(* Logix 5000 project; controller QW361 vendor 1 type 14 code 107 rev 32.11; software revision 32.00; part 8 of 20 *)

        [856].log_data[0].maxminute := 50, [856].log_data[0].valid := 1, [856].log_data[1].valid := 1, [856].log_data[2].valid := 1, [856].log_data[3].valid := 1, [856].log_data[4].valid := 1, [856].time.Year := 2022, [856].time.Month := 4, [856].time.Day := 26, [856].time.Hour := 20, [856].time.Minute := 54, [856].time.Second := 59, [856].time.DST_ON := 1, [857].log_data[0].min := 1.0, [857].log_data[0].max := 1.0, [857].log_data[0].total := 299.999, [857].log_data[0].time := 299.999, [857].log_data[0].minminute := 55, [857].log_data[0].maxminute := 55, [857].log_data[0].valid := 1, [857].log_data[1].valid := 1, [857].log_data[2].valid := 1, [857].log_data[3].valid := 1, [857].log_data[4].valid := 1, [857].time.Year := 2022, [857].time.Month := 4, [857].time.Day := 26, [857].time.Hour := 20, [857].time.Minute := 59, [857].time.Second := 59, [857].time.DST_ON := 1, [858].log_data[0].min := 1.0, [858].log_data[0].max := 1.0, [858].log_data[0].total := 300.0, [858].log_data[0].time := 300.0, [858].log_data[0].valid := 1, [858].log_data[1].valid := 1, [858].log_data[2].valid := 1, [858].log_data[3].valid := 1, [858].log_data[4].valid := 1, [858].time.Year := 2022, [858].time.Month := 4, [858].time.Day := 26, [858].time.Hour := 21, [858].time.Minute := 4, [858].time.Second := 59, [858].time.DST_ON := 1, [859].log_data[0].min := 1.0, [859].log_data[0].max := 1.0, [859].log_data[0].total := 300.0, [859].log_data[0].time := 300.0, [859].log_data[0].minminute := 5, [859].log_data[0].maxminute := 5, [859].log_data[0].valid := 1, [859].log_data[1].valid := 1, [859].log_data[2].valid := 1, [859].log_data[3].valid := 1, [859].log_data[4].valid := 1, [859].time.Year := 2022, [859].time.Month := 4,
        [859].time.Day := 26, [859].time.Hour := 21, [859].time.Minute := 9, [859].time.Second := 59, [859].time.DST_ON := 1, [860].log_data[0].min := 1.0, [860].log_data[0].max := 1.0, [860].log_data[0].total := 300.0, [860].log_data[0].time := 300.0, [860].log_data[0].minminute := 10, [860].log_data[0].maxminute := 10, [860].log_data[0].valid := 1, [860].log_data[1].valid := 1, [860].log_data[2].valid := 1, [860].log_data[3].valid := 1, [860].log_data[4].valid := 1, [860].time.Year := 2022, [860].time.Month := 4, [860].time.Day := 26, [860].time.Hour := 21, [860].time.Minute := 14, [860].time.Second := 59, [860].time.DST_ON := 1, [861].log_data[0].min := 1.0, [861].log_data[0].max := 1.0, [861].log_data[0].total := 300.0, [861].log_data[0].time := 300.0, [861].log_data[0].minminute := 15, [861].log_data[0].maxminute := 15, [861].log_data[0].valid := 1, [861].log_data[1].valid := 1, [861].log_data[2].valid := 1, [861].log_data[3].valid := 1, [861].log_data[4].valid := 1, [861].time.Year := 2022, [861].time.Month := 4, [861].time.Day := 26, [861].time.Hour := 21, [861].time.Minute := 19, [861].time.Second := 59, [861].time.DST_ON := 1, [862].log_data[0].min := 1.0, [862].log_data[0].max := 1.0, [862].log_data[0].total := 300.0, [862].log_data[0].time := 300.0, [862].log_data[0].minminute := 20, [862].log_data[0].maxminute := 20, [862].log_data[0].valid := 1, [862].log_data[1].valid := 1, [862].log_data[2].valid := 1, [862].log_data[3].valid := 1, [862].log_data[4].valid := 1, [862].time.Year := 2022, [862].time.Month := 4, [862].time.Day := 26, [862].time.Hour := 21, [862].time.Minute := 24, [862].time.Second := 59, [862].time.DST_ON := 1, [863].log_data[0].min := 1.0,
        [863].log_data[0].max := 1.0, [863].log_data[0].total := 300.0, [863].log_data[0].time := 300.0, [863].log_data[0].minminute := 25, [863].log_data[0].maxminute := 25, [863].log_data[0].valid := 1, [863].log_data[1].valid := 1, [863].log_data[2].valid := 1, [863].log_data[3].valid := 1, [863].log_data[4].valid := 1, [863].time.Year := 2022, [863].time.Month := 4, [863].time.Day := 26, [863].time.Hour := 21, [863].time.Minute := 29, [863].time.Second := 59, [863].time.DST_ON := 1, [864].log_data[0].min := 1.0, [864].log_data[0].max := 1.0, [864].log_data[0].total := 300.0, [864].log_data[0].time := 300.0, [864].log_data[0].minminute := 30, [864].log_data[0].maxminute := 30, [864].log_data[0].valid := 1, [864].log_data[1].valid := 1, [864].log_data[2].valid := 1, [864].log_data[3].valid := 1, [864].log_data[4].valid := 1, [864].time.Year := 2022, [864].time.Month := 4, [864].time.Day := 26, [864].time.Hour := 21, [864].time.Minute := 34, [864].time.Second := 59, [864].time.DST_ON := 1, [865].log_data[0].min := 1.0, [865].log_data[0].max := 1.0, [865].log_data[0].total := 300.0, [865].log_data[0].time := 300.0, [865].log_data[0].minminute := 35, [865].log_data[0].maxminute := 35, [865].log_data[0].valid := 1, [865].log_data[1].valid := 1, [865].log_data[2].valid := 1, [865].log_data[3].valid := 1, [865].log_data[4].valid := 1, [865].time.Year := 2022, [865].time.Month := 4, [865].time.Day := 26, [865].time.Hour := 21, [865].time.Minute := 39, [865].time.Second := 59, [865].time.DST_ON := 1, [866].log_data[0].min := 1.0, [866].log_data[0].max := 1.0, [866].log_data[0].total := 300.0, [866].log_data[0].time := 300.0, [866].log_data[0].minminute := 40, [866].log_data[0].maxminute := 40, [866].log_data[0].valid := 1,
        [866].log_data[1].valid := 1, [866].log_data[2].valid := 1, [866].log_data[3].valid := 1, [866].log_data[4].valid := 1, [866].time.Year := 2022, [866].time.Month := 4, [866].time.Day := 26, [866].time.Hour := 21, [866].time.Minute := 44, [866].time.Second := 59, [866].time.DST_ON := 1, [867].log_data[0].min := 1.0, [867].log_data[0].max := 1.0, [867].log_data[0].total := 300.0, [867].log_data[0].time := 300.0, [867].log_data[0].minminute := 45, [867].log_data[0].maxminute := 45, [867].log_data[0].valid := 1, [867].log_data[1].valid := 1, [867].log_data[2].valid := 1, [867].log_data[3].valid := 1, [867].log_data[4].valid := 1, [867].time.Year := 2022, [867].time.Month := 4, [867].time.Day := 26, [867].time.Hour := 21, [867].time.Minute := 49, [867].time.Second := 59, [867].time.DST_ON := 1, [868].log_data[0].min := 1.0, [868].log_data[0].max := 1.0, [868].log_data[0].total := 300.0, [868].log_data[0].time := 300.0, [868].log_data[0].minminute := 50, [868].log_data[0].maxminute := 50, [868].log_data[0].valid := 1, [868].log_data[1].valid := 1, [868].log_data[2].valid := 1, [868].log_data[3].valid := 1, [868].log_data[4].valid := 1, [868].time.Year := 2022, [868].time.Month := 4, [868].time.Day := 26, [868].time.Hour := 21, [868].time.Minute := 54, [868].time.Second := 59, [868].time.DST_ON := 1, [869].log_data[0].min := 1.0, [869].log_data[0].max := 1.0, [869].log_data[0].total := 300.0, [869].log_data[0].time := 300.0, [869].log_data[0].minminute := 55, [869].log_data[0].maxminute := 55, [869].log_data[0].valid := 1, [869].log_data[1].valid := 1, [869].log_data[2].valid := 1, [869].log_data[3].valid := 1, [869].log_data[4].valid := 1, [869].time.Year := 2022, [869].time.Month := 4,
        [869].time.Day := 26, [869].time.Hour := 21, [869].time.Minute := 59, [869].time.Second := 59, [869].time.DST_ON := 1, [870].log_data[0].min := 1.0, [870].log_data[0].max := 1.0, [870].log_data[0].total := 300.0, [870].log_data[0].time := 300.0, [870].log_data[0].valid := 1, [870].log_data[1].valid := 1, [870].log_data[2].valid := 1, [870].log_data[3].valid := 1, [870].log_data[4].valid := 1, [870].time.Year := 2022, [870].time.Month := 4, [870].time.Day := 26, [870].time.Hour := 22, [870].time.Minute := 4, [870].time.Second := 59, [870].time.DST_ON := 1, [871].log_data[0].min := 1.0, [871].log_data[0].max := 1.0, [871].log_data[0].total := 300.0, [871].log_data[0].time := 300.0, [871].log_data[0].minminute := 5, [871].log_data[0].maxminute := 5, [871].log_data[0].valid := 1, [871].log_data[1].valid := 1, [871].log_data[2].valid := 1, [871].log_data[3].valid := 1, [871].log_data[4].valid := 1, [871].time.Year := 2022, [871].time.Month := 4, [871].time.Day := 26, [871].time.Hour := 22, [871].time.Minute := 9, [871].time.Second := 59, [871].time.DST_ON := 1, [872].log_data[0].min := 1.0, [872].log_data[0].max := 1.0, [872].log_data[0].total := 300.0, [872].log_data[0].time := 300.0, [872].log_data[0].minminute := 10, [872].log_data[0].maxminute := 10, [872].log_data[0].valid := 1, [872].log_data[1].valid := 1, [872].log_data[2].valid := 1, [872].log_data[3].valid := 1, [872].log_data[4].valid := 1, [872].time.Year := 2022, [872].time.Month := 4, [872].time.Day := 26, [872].time.Hour := 22, [872].time.Minute := 14, [872].time.Second := 59, [872].time.DST_ON := 1, [873].log_data[0].min := 1.0, [873].log_data[0].max := 1.0, [873].log_data[0].total := 300.0,
        [873].log_data[0].time := 300.0, [873].log_data[0].minminute := 15, [873].log_data[0].maxminute := 15, [873].log_data[0].valid := 1, [873].log_data[1].valid := 1, [873].log_data[2].valid := 1, [873].log_data[3].valid := 1, [873].log_data[4].valid := 1, [873].time.Year := 2022, [873].time.Month := 4, [873].time.Day := 26, [873].time.Hour := 22, [873].time.Minute := 19, [873].time.Second := 59, [873].time.DST_ON := 1, [874].log_data[0].min := 1.0, [874].log_data[0].max := 1.0, [874].log_data[0].total := 300.0, [874].log_data[0].time := 300.0, [874].log_data[0].minminute := 20, [874].log_data[0].maxminute := 20, [874].log_data[0].valid := 1, [874].log_data[1].valid := 1, [874].log_data[2].valid := 1, [874].log_data[3].valid := 1, [874].log_data[4].valid := 1, [874].time.Year := 2022, [874].time.Month := 4, [874].time.Day := 26, [874].time.Hour := 22, [874].time.Minute := 24, [874].time.Second := 59, [874].time.DST_ON := 1, [875].log_data[0].min := 1.0, [875].log_data[0].max := 1.0, [875].log_data[0].total := 300.0, [875].log_data[0].time := 300.0, [875].log_data[0].minminute := 25, [875].log_data[0].maxminute := 25, [875].log_data[0].valid := 1, [875].log_data[1].valid := 1, [875].log_data[2].valid := 1, [875].log_data[3].valid := 1, [875].log_data[4].valid := 1, [875].time.Year := 2022, [875].time.Month := 4, [875].time.Day := 26, [875].time.Hour := 22, [875].time.Minute := 29, [875].time.Second := 59, [875].time.DST_ON := 1, [876].log_data[0].min := 1.0, [876].log_data[0].max := 1.0, [876].log_data[0].total := 300.0, [876].log_data[0].time := 300.0, [876].log_data[0].minminute := 30, [876].log_data[0].maxminute := 30, [876].log_data[0].valid := 1, [876].log_data[1].valid := 1, [876].log_data[2].valid := 1,
        [876].log_data[3].valid := 1, [876].log_data[4].valid := 1, [876].time.Year := 2022, [876].time.Month := 4, [876].time.Day := 26, [876].time.Hour := 22, [876].time.Minute := 34, [876].time.Second := 59, [876].time.DST_ON := 1, [877].log_data[0].min := 1.0, [877].log_data[0].max := 1.0, [877].log_data[0].total := 300.0, [877].log_data[0].time := 300.0, [877].log_data[0].minminute := 35, [877].log_data[0].maxminute := 35, [877].log_data[0].valid := 1, [877].log_data[1].valid := 1, [877].log_data[2].valid := 1, [877].log_data[3].valid := 1, [877].log_data[4].valid := 1, [877].time.Year := 2022, [877].time.Month := 4, [877].time.Day := 26, [877].time.Hour := 22, [877].time.Minute := 39, [877].time.Second := 59, [877].time.DST_ON := 1, [878].log_data[0].min := 1.0, [878].log_data[0].max := 1.0, [878].log_data[0].total := 300.0, [878].log_data[0].time := 300.0, [878].log_data[0].minminute := 40, [878].log_data[0].maxminute := 40, [878].log_data[0].valid := 1, [878].log_data[1].valid := 1, [878].log_data[2].valid := 1, [878].log_data[3].valid := 1, [878].log_data[4].valid := 1, [878].time.Year := 2022, [878].time.Month := 4, [878].time.Day := 26, [878].time.Hour := 22, [878].time.Minute := 44, [878].time.Second := 59, [878].time.DST_ON := 1, [879].log_data[0].min := 1.0, [879].log_data[0].max := 1.0, [879].log_data[0].total := 300.0, [879].log_data[0].time := 300.0, [879].log_data[0].minminute := 45, [879].log_data[0].maxminute := 45, [879].log_data[0].valid := 1, [879].log_data[1].valid := 1, [879].log_data[2].valid := 1, [879].log_data[3].valid := 1, [879].log_data[4].valid := 1, [879].time.Year := 2022, [879].time.Month := 4, [879].time.Day := 26, [879].time.Hour := 22,
        [879].time.Minute := 49, [879].time.Second := 59, [879].time.DST_ON := 1, [880].log_data[0].min := 1.0, [880].log_data[0].max := 1.0, [880].log_data[0].total := 300.0, [880].log_data[0].time := 300.0, [880].log_data[0].minminute := 50, [880].log_data[0].maxminute := 50, [880].log_data[0].valid := 1, [880].log_data[1].valid := 1, [880].log_data[2].valid := 1, [880].log_data[3].valid := 1, [880].log_data[4].valid := 1, [880].time.Year := 2022, [880].time.Month := 4, [880].time.Day := 26, [880].time.Hour := 22, [880].time.Minute := 54, [880].time.Second := 59, [880].time.DST_ON := 1, [881].log_data[0].min := 1.0, [881].log_data[0].max := 1.0, [881].log_data[0].total := 300.0, [881].log_data[0].time := 300.0, [881].log_data[0].minminute := 55, [881].log_data[0].maxminute := 55, [881].log_data[0].valid := 1, [881].log_data[1].valid := 1, [881].log_data[2].valid := 1, [881].log_data[3].valid := 1, [881].log_data[4].valid := 1, [881].time.Year := 2022, [881].time.Month := 4, [881].time.Day := 26, [881].time.Hour := 22, [881].time.Minute := 59, [881].time.Second := 59, [881].time.DST_ON := 1, [882].log_data[0].min := 1.0, [882].log_data[0].max := 1.0, [882].log_data[0].total := 300.0, [882].log_data[0].time := 300.0, [882].log_data[0].valid := 1, [882].log_data[1].valid := 1, [882].log_data[2].valid := 1, [882].log_data[3].valid := 1, [882].log_data[4].valid := 1, [882].time.Year := 2022, [882].time.Month := 4, [882].time.Day := 26, [882].time.Hour := 23, [882].time.Minute := 4, [882].time.Second := 59, [882].time.DST_ON := 1, [883].log_data[0].min := 1.0, [883].log_data[0].max := 1.0, [883].log_data[0].total := 300.0, [883].log_data[0].time := 300.0, [883].log_data[0].minminute := 5,
        [883].log_data[0].maxminute := 5, [883].log_data[0].valid := 1, [883].log_data[1].valid := 1, [883].log_data[2].valid := 1, [883].log_data[3].valid := 1, [883].log_data[4].valid := 1, [883].time.Year := 2022, [883].time.Month := 4, [883].time.Day := 26, [883].time.Hour := 23, [883].time.Minute := 9, [883].time.Second := 59, [883].time.DST_ON := 1, [884].log_data[0].min := 1.0, [884].log_data[0].max := 1.0, [884].log_data[0].total := 300.0, [884].log_data[0].time := 300.0, [884].log_data[0].minminute := 10, [884].log_data[0].maxminute := 10, [884].log_data[0].valid := 1, [884].log_data[1].valid := 1, [884].log_data[2].valid := 1, [884].log_data[3].valid := 1, [884].log_data[4].valid := 1, [884].time.Year := 2022, [884].time.Month := 4, [884].time.Day := 26, [884].time.Hour := 23, [884].time.Minute := 14, [884].time.Second := 59, [884].time.DST_ON := 1, [885].log_data[0].min := 1.0, [885].log_data[0].max := 1.0, [885].log_data[0].total := 300.0, [885].log_data[0].time := 300.0, [885].log_data[0].minminute := 15, [885].log_data[0].maxminute := 15, [885].log_data[0].valid := 1, [885].log_data[1].valid := 1, [885].log_data[2].valid := 1, [885].log_data[3].valid := 1, [885].log_data[4].valid := 1, [885].time.Year := 2022, [885].time.Month := 4, [885].time.Day := 26, [885].time.Hour := 23, [885].time.Minute := 19, [885].time.Second := 59, [885].time.DST_ON := 1, [886].log_data[0].min := 1.0, [886].log_data[0].max := 1.0, [886].log_data[0].total := 300.0, [886].log_data[0].time := 300.0, [886].log_data[0].minminute := 20, [886].log_data[0].maxminute := 20, [886].log_data[0].valid := 1, [886].log_data[1].valid := 1, [886].log_data[2].valid := 1, [886].log_data[3].valid := 1, [886].log_data[4].valid := 1,
        [886].time.Year := 2022, [886].time.Month := 4, [886].time.Day := 26, [886].time.Hour := 23, [886].time.Minute := 24, [886].time.Second := 59, [886].time.DST_ON := 1, [887].log_data[0].min := 1.0, [887].log_data[0].max := 1.0, [887].log_data[0].total := 300.0, [887].log_data[0].time := 300.0, [887].log_data[0].minminute := 25, [887].log_data[0].maxminute := 25, [887].log_data[0].valid := 1, [887].log_data[1].valid := 1, [887].log_data[2].valid := 1, [887].log_data[3].valid := 1, [887].log_data[4].valid := 1, [887].time.Year := 2022, [887].time.Month := 4, [887].time.Day := 26, [887].time.Hour := 23, [887].time.Minute := 29, [887].time.Second := 59, [887].time.DST_ON := 1, [888].log_data[0].min := 1.0, [888].log_data[0].max := 1.0, [888].log_data[0].total := 300.0, [888].log_data[0].time := 300.0, [888].log_data[0].minminute := 30, [888].log_data[0].maxminute := 30, [888].log_data[0].valid := 1, [888].log_data[1].valid := 1, [888].log_data[2].valid := 1, [888].log_data[3].valid := 1, [888].log_data[4].valid := 1, [888].time.Year := 2022, [888].time.Month := 4, [888].time.Day := 26, [888].time.Hour := 23, [888].time.Minute := 34, [888].time.Second := 59, [888].time.DST_ON := 1, [889].log_data[0].min := 1.0, [889].log_data[0].max := 1.0, [889].log_data[0].total := 300.0, [889].log_data[0].time := 300.0, [889].log_data[0].minminute := 35, [889].log_data[0].maxminute := 35, [889].log_data[0].valid := 1, [889].log_data[1].valid := 1, [889].log_data[2].valid := 1, [889].log_data[3].valid := 1, [889].log_data[4].valid := 1, [889].time.Year := 2022, [889].time.Month := 4, [889].time.Day := 26, [889].time.Hour := 23, [889].time.Minute := 39, [889].time.Second := 59,
        [889].time.DST_ON := 1, [890].log_data[0].min := 1.0, [890].log_data[0].max := 1.0, [890].log_data[0].total := 300.0, [890].log_data[0].time := 300.0, [890].log_data[0].minminute := 40, [890].log_data[0].maxminute := 40, [890].log_data[0].valid := 1, [890].log_data[1].valid := 1, [890].log_data[2].valid := 1, [890].log_data[3].valid := 1, [890].log_data[4].valid := 1, [890].time.Year := 2022, [890].time.Month := 4, [890].time.Day := 26, [890].time.Hour := 23, [890].time.Minute := 44, [890].time.Second := 59, [890].time.DST_ON := 1, [891].log_data[0].min := 1.0, [891].log_data[0].max := 1.0, [891].log_data[0].total := 300.0, [891].log_data[0].time := 300.0, [891].log_data[0].minminute := 45, [891].log_data[0].maxminute := 45, [891].log_data[0].valid := 1, [891].log_data[1].valid := 1, [891].log_data[2].valid := 1, [891].log_data[3].valid := 1, [891].log_data[4].valid := 1, [891].time.Year := 2022, [891].time.Month := 4, [891].time.Day := 26, [891].time.Hour := 23, [891].time.Minute := 49, [891].time.Second := 59, [891].time.DST_ON := 1, [892].log_data[0].min := 1.0, [892].log_data[0].max := 1.0, [892].log_data[0].total := 300.0, [892].log_data[0].time := 300.0, [892].log_data[0].minminute := 50, [892].log_data[0].maxminute := 50, [892].log_data[0].valid := 1, [892].log_data[1].valid := 1, [892].log_data[2].valid := 1, [892].log_data[3].valid := 1, [892].log_data[4].valid := 1, [892].time.Year := 2022, [892].time.Month := 4, [892].time.Day := 26, [892].time.Hour := 23, [892].time.Minute := 54, [892].time.Second := 59, [892].time.DST_ON := 1, [893].log_data[0].min := 1.0, [893].log_data[0].max := 1.0, [893].log_data[0].total := 299.999, [893].log_data[0].time := 299.999, [893].log_data[0].minminute := 55,
        [893].log_data[0].maxminute := 55, [893].log_data[0].valid := 1, [893].log_data[1].valid := 1, [893].log_data[2].valid := 1, [893].log_data[3].valid := 1, [893].log_data[4].valid := 1, [893].time.Year := 2022, [893].time.Month := 4, [893].time.Day := 26, [893].time.Hour := 23, [893].time.Minute := 59, [893].time.Second := 59, [893].time.DST_ON := 1, [894].log_data[0].min := 1.0, [894].log_data[0].max := 1.0, [894].log_data[0].total := 300.0, [894].log_data[0].time := 300.0, [894].log_data[0].valid := 1, [894].log_data[1].valid := 1, [894].log_data[2].valid := 1, [894].log_data[3].valid := 1, [894].log_data[4].valid := 1, [894].time.Year := 2022, [894].time.Month := 4, [894].time.Day := 27, [894].time.Minute := 4, [894].time.Second := 59, [894].time.DST_ON := 1, [895].log_data[0].min := 1.0, [895].log_data[0].max := 1.0, [895].log_data[0].total := 300.0, [895].log_data[0].time := 300.0, [895].log_data[0].minminute := 5, [895].log_data[0].maxminute := 5, [895].log_data[0].valid := 1, [895].log_data[1].valid := 1, [895].log_data[2].valid := 1, [895].log_data[3].valid := 1, [895].log_data[4].valid := 1, [895].time.Year := 2022, [895].time.Month := 4, [895].time.Day := 27, [895].time.Minute := 9, [895].time.Second := 59, [895].time.DST_ON := 1, [896].log_data[0].min := 1.0, [896].log_data[0].max := 1.0, [896].log_data[0].total := 300.0, [896].log_data[0].time := 300.0, [896].log_data[0].minminute := 10, [896].log_data[0].maxminute := 10, [896].log_data[0].valid := 1, [896].log_data[1].valid := 1, [896].log_data[2].valid := 1, [896].log_data[3].valid := 1, [896].log_data[4].valid := 1, [896].time.Year := 2022, [896].time.Month := 4, [896].time.Day := 27, [896].time.Minute := 14,
        [896].time.Second := 59, [896].time.DST_ON := 1, [897].log_data[0].min := 1.0, [897].log_data[0].max := 1.0, [897].log_data[0].total := 300.0, [897].log_data[0].time := 300.0, [897].log_data[0].minminute := 15, [897].log_data[0].maxminute := 15, [897].log_data[0].valid := 1, [897].log_data[1].valid := 1, [897].log_data[2].valid := 1, [897].log_data[3].valid := 1, [897].log_data[4].valid := 1, [897].time.Year := 2022, [897].time.Month := 4, [897].time.Day := 27, [897].time.Minute := 19, [897].time.Second := 59, [897].time.DST_ON := 1, [898].log_data[0].min := 1.0, [898].log_data[0].max := 1.0, [898].log_data[0].total := 300.0, [898].log_data[0].time := 300.0, [898].log_data[0].minminute := 20, [898].log_data[0].maxminute := 20, [898].log_data[0].valid := 1, [898].log_data[1].valid := 1, [898].log_data[2].valid := 1, [898].log_data[3].valid := 1, [898].log_data[4].valid := 1, [898].time.Year := 2022, [898].time.Month := 4, [898].time.Day := 27, [898].time.Minute := 24, [898].time.Second := 59, [898].time.DST_ON := 1, [899].log_data[0].min := 1.0, [899].log_data[0].max := 1.0, [899].log_data[0].total := 300.0, [899].log_data[0].time := 300.0, [899].log_data[0].minminute := 25, [899].log_data[0].maxminute := 25, [899].log_data[0].valid := 1, [899].log_data[1].valid := 1, [899].log_data[2].valid := 1, [899].log_data[3].valid := 1, [899].log_data[4].valid := 1, [899].time.Year := 2022, [899].time.Month := 4, [899].time.Day := 27, [899].time.Minute := 29, [899].time.Second := 59, [899].time.DST_ON := 1, [900].log_data[0].min := 1.0, [900].log_data[0].max := 1.0, [900].log_data[0].total := 300.0, [900].log_data[0].time := 300.0, [900].log_data[0].minminute := 30, [900].log_data[0].maxminute := 30, [900].log_data[0].valid := 1,
        [900].log_data[1].valid := 1, [900].log_data[2].valid := 1, [900].log_data[3].valid := 1, [900].log_data[4].valid := 1, [900].time.Year := 2022, [900].time.Month := 4, [900].time.Day := 27, [900].time.Minute := 34, [900].time.Second := 59, [900].time.DST_ON := 1, [901].log_data[0].min := 1.0, [901].log_data[0].max := 1.0, [901].log_data[0].total := 300.0, [901].log_data[0].time := 300.0, [901].log_data[0].minminute := 35, [901].log_data[0].maxminute := 35, [901].log_data[0].valid := 1, [901].log_data[1].valid := 1, [901].log_data[2].valid := 1, [901].log_data[3].valid := 1, [901].log_data[4].valid := 1, [901].time.Year := 2022, [901].time.Month := 4, [901].time.Day := 27, [901].time.Minute := 39, [901].time.Second := 59, [901].time.DST_ON := 1, [902].log_data[0].min := 1.0, [902].log_data[0].max := 1.0, [902].log_data[0].total := 300.0, [902].log_data[0].time := 300.0, [902].log_data[0].minminute := 40, [902].log_data[0].maxminute := 40, [902].log_data[0].valid := 1, [902].log_data[1].valid := 1, [902].log_data[2].valid := 1, [902].log_data[3].valid := 1, [902].log_data[4].valid := 1, [902].time.Year := 2022, [902].time.Month := 4, [902].time.Day := 27, [902].time.Minute := 44, [902].time.Second := 59, [902].time.DST_ON := 1, [903].log_data[0].min := 1.0, [903].log_data[0].max := 1.0, [903].log_data[0].total := 300.0, [903].log_data[0].time := 300.0, [903].log_data[0].minminute := 45, [903].log_data[0].maxminute := 45, [903].log_data[0].valid := 1, [903].log_data[1].valid := 1, [903].log_data[2].valid := 1, [903].log_data[3].valid := 1, [903].log_data[4].valid := 1, [903].time.Year := 2022, [903].time.Month := 4, [903].time.Day := 27, [903].time.Minute := 49, [903].time.Second := 59,
        [903].time.DST_ON := 1, [904].log_data[0].min := 1.0, [904].log_data[0].max := 1.0, [904].log_data[0].total := 300.0, [904].log_data[0].time := 300.0, [904].log_data[0].minminute := 50, [904].log_data[0].maxminute := 50, [904].log_data[0].valid := 1, [904].log_data[1].valid := 1, [904].log_data[2].valid := 1, [904].log_data[3].valid := 1, [904].log_data[4].valid := 1, [904].time.Year := 2022, [904].time.Month := 4, [904].time.Day := 27, [904].time.Minute := 54, [904].time.Second := 59, [904].time.DST_ON := 1, [905].log_data[0].min := 1.0, [905].log_data[0].max := 1.0, [905].log_data[0].total := 300.0, [905].log_data[0].time := 300.0, [905].log_data[0].minminute := 55, [905].log_data[0].maxminute := 55, [905].log_data[0].valid := 1, [905].log_data[1].valid := 1, [905].log_data[2].valid := 1, [905].log_data[3].valid := 1, [905].log_data[4].valid := 1, [905].time.Year := 2022, [905].time.Month := 4, [905].time.Day := 27, [905].time.Minute := 59, [905].time.Second := 59, [905].time.DST_ON := 1, [906].log_data[0].min := 1.0, [906].log_data[0].max := 1.0, [906].log_data[0].total := 300.0, [906].log_data[0].time := 300.0, [906].log_data[0].valid := 1, [906].log_data[1].valid := 1, [906].log_data[2].valid := 1, [906].log_data[3].valid := 1, [906].log_data[4].valid := 1, [906].time.Year := 2022, [906].time.Month := 4, [906].time.Day := 27, [906].time.Hour := 1, [906].time.Minute := 4, [906].time.Second := 59, [906].time.DST_ON := 1, [907].log_data[0].min := 1.0, [907].log_data[0].max := 1.0, [907].log_data[0].total := 300.0, [907].log_data[0].time := 300.0, [907].log_data[0].minminute := 5, [907].log_data[0].maxminute := 5, [907].log_data[0].valid := 1, [907].log_data[1].valid := 1, [907].log_data[2].valid := 1,
        [907].log_data[3].valid := 1, [907].log_data[4].valid := 1, [907].time.Year := 2022, [907].time.Month := 4, [907].time.Day := 27, [907].time.Hour := 1, [907].time.Minute := 9, [907].time.Second := 59, [907].time.DST_ON := 1, [908].log_data[0].min := 1.0, [908].log_data[0].max := 1.0, [908].log_data[0].total := 300.0, [908].log_data[0].time := 300.0, [908].log_data[0].minminute := 10, [908].log_data[0].maxminute := 10, [908].log_data[0].valid := 1, [908].log_data[1].valid := 1, [908].log_data[2].valid := 1, [908].log_data[3].valid := 1, [908].log_data[4].valid := 1, [908].time.Year := 2022, [908].time.Month := 4, [908].time.Day := 27, [908].time.Hour := 1, [908].time.Minute := 14, [908].time.Second := 59, [908].time.DST_ON := 1, [909].log_data[0].min := 1.0, [909].log_data[0].max := 1.0, [909].log_data[0].total := 300.0, [909].log_data[0].time := 300.0, [909].log_data[0].minminute := 15, [909].log_data[0].maxminute := 15, [909].log_data[0].valid := 1, [909].log_data[1].valid := 1, [909].log_data[2].valid := 1, [909].log_data[3].valid := 1, [909].log_data[4].valid := 1, [909].time.Year := 2022, [909].time.Month := 4, [909].time.Day := 27, [909].time.Hour := 1, [909].time.Minute := 19, [909].time.Second := 59, [909].time.DST_ON := 1, [910].log_data[0].min := 1.0, [910].log_data[0].max := 1.0, [910].log_data[0].total := 300.0, [910].log_data[0].time := 300.0, [910].log_data[0].minminute := 20, [910].log_data[0].maxminute := 20, [910].log_data[0].valid := 1, [910].log_data[1].valid := 1, [910].log_data[2].valid := 1, [910].log_data[3].valid := 1, [910].log_data[4].valid := 1, [910].time.Year := 2022, [910].time.Month := 4, [910].time.Day := 27, [910].time.Hour := 1,
        [910].time.Minute := 24, [910].time.Second := 59, [910].time.DST_ON := 1, [911].log_data[0].min := 1.0, [911].log_data[0].max := 1.0, [911].log_data[0].total := 300.0, [911].log_data[0].time := 300.0, [911].log_data[0].minminute := 25, [911].log_data[0].maxminute := 25, [911].log_data[0].valid := 1, [911].log_data[1].valid := 1, [911].log_data[2].valid := 1, [911].log_data[3].valid := 1, [911].log_data[4].valid := 1, [911].time.Year := 2022, [911].time.Month := 4, [911].time.Day := 27, [911].time.Hour := 1, [911].time.Minute := 29, [911].time.Second := 59, [911].time.DST_ON := 1, [912].log_data[0].min := 1.0, [912].log_data[0].max := 1.0, [912].log_data[0].total := 300.0, [912].log_data[0].time := 300.0, [912].log_data[0].minminute := 30, [912].log_data[0].maxminute := 30, [912].log_data[0].valid := 1, [912].log_data[1].valid := 1, [912].log_data[2].valid := 1, [912].log_data[3].valid := 1, [912].log_data[4].valid := 1, [912].time.Year := 2022, [912].time.Month := 4, [912].time.Day := 27, [912].time.Hour := 1, [912].time.Minute := 34, [912].time.Second := 59, [912].time.DST_ON := 1, [913].log_data[0].min := 1.0, [913].log_data[0].max := 1.0, [913].log_data[0].total := 300.0, [913].log_data[0].time := 300.0, [913].log_data[0].minminute := 35, [913].log_data[0].maxminute := 35, [913].log_data[0].valid := 1, [913].log_data[1].valid := 1, [913].log_data[2].valid := 1, [913].log_data[3].valid := 1, [913].log_data[4].valid := 1, [913].time.Year := 2022, [913].time.Month := 4, [913].time.Day := 27, [913].time.Hour := 1, [913].time.Minute := 39, [913].time.Second := 59, [913].time.DST_ON := 1, [914].log_data[0].min := 1.0, [914].log_data[0].max := 1.0, [914].log_data[0].total := 300.0,
        [914].log_data[0].time := 300.0, [914].log_data[0].minminute := 40, [914].log_data[0].maxminute := 40, [914].log_data[0].valid := 1, [914].log_data[1].valid := 1, [914].log_data[2].valid := 1, [914].log_data[3].valid := 1, [914].log_data[4].valid := 1, [914].time.Year := 2022, [914].time.Month := 4, [914].time.Day := 27, [914].time.Hour := 1, [914].time.Minute := 44, [914].time.Second := 59, [914].time.DST_ON := 1, [915].log_data[0].min := 1.0, [915].log_data[0].max := 1.0, [915].log_data[0].total := 300.0, [915].log_data[0].time := 300.0, [915].log_data[0].minminute := 45, [915].log_data[0].maxminute := 45, [915].log_data[0].valid := 1, [915].log_data[1].valid := 1, [915].log_data[2].valid := 1, [915].log_data[3].valid := 1, [915].log_data[4].valid := 1, [915].time.Year := 2022, [915].time.Month := 4, [915].time.Day := 27, [915].time.Hour := 1, [915].time.Minute := 49, [915].time.Second := 59, [915].time.DST_ON := 1, [916].log_data[0].min := 1.0, [916].log_data[0].max := 1.0, [916].log_data[0].total := 300.0, [916].log_data[0].time := 300.0, [916].log_data[0].minminute := 50, [916].log_data[0].maxminute := 50, [916].log_data[0].valid := 1, [916].log_data[1].valid := 1, [916].log_data[2].valid := 1, [916].log_data[3].valid := 1, [916].log_data[4].valid := 1, [916].time.Year := 2022, [916].time.Month := 4, [916].time.Day := 27, [916].time.Hour := 1, [916].time.Minute := 54, [916].time.Second := 59, [916].time.DST_ON := 1, [917].log_data[0].min := 1.0, [917].log_data[0].max := 1.0, [917].log_data[0].total := 300.0, [917].log_data[0].time := 300.0, [917].log_data[0].minminute := 55, [917].log_data[0].maxminute := 55, [917].log_data[0].valid := 1, [917].log_data[1].valid := 1, [917].log_data[2].valid := 1,
        [917].log_data[3].valid := 1, [917].log_data[4].valid := 1, [917].time.Year := 2022, [917].time.Month := 4, [917].time.Day := 27, [917].time.Hour := 1, [917].time.Minute := 59, [917].time.Second := 59, [917].time.DST_ON := 1, [918].log_data[0].min := 1.0, [918].log_data[0].max := 1.0, [918].log_data[0].total := 300.0, [918].log_data[0].time := 300.0, [918].log_data[0].valid := 1, [918].log_data[1].valid := 1, [918].log_data[2].valid := 1, [918].log_data[3].valid := 1, [918].log_data[4].valid := 1, [918].time.Year := 2022, [918].time.Month := 4, [918].time.Day := 27, [918].time.Hour := 2, [918].time.Minute := 4, [918].time.Second := 59, [918].time.DST_ON := 1, [919].log_data[0].min := 1.0, [919].log_data[0].max := 1.0, [919].log_data[0].total := 300.0, [919].log_data[0].time := 300.0, [919].log_data[0].minminute := 5, [919].log_data[0].maxminute := 5, [919].log_data[0].valid := 1, [919].log_data[1].valid := 1, [919].log_data[2].valid := 1, [919].log_data[3].valid := 1, [919].log_data[4].valid := 1, [919].time.Year := 2022, [919].time.Month := 4, [919].time.Day := 27, [919].time.Hour := 2, [919].time.Minute := 9, [919].time.Second := 59, [919].time.DST_ON := 1, [920].log_data[0].min := 1.0, [920].log_data[0].max := 1.0, [920].log_data[0].total := 300.0, [920].log_data[0].time := 300.0, [920].log_data[0].minminute := 10, [920].log_data[0].maxminute := 10, [920].log_data[0].valid := 1, [920].log_data[1].valid := 1, [920].log_data[2].valid := 1, [920].log_data[3].valid := 1, [920].log_data[4].valid := 1, [920].time.Year := 2022, [920].time.Month := 4, [920].time.Day := 27, [920].time.Hour := 2, [920].time.Minute := 14, [920].time.Second := 59,
        [920].time.DST_ON := 1, [921].log_data[0].min := 1.0, [921].log_data[0].max := 1.0, [921].log_data[0].total := 300.0, [921].log_data[0].time := 300.0, [921].log_data[0].minminute := 15, [921].log_data[0].maxminute := 15, [921].log_data[0].valid := 1, [921].log_data[1].valid := 1, [921].log_data[2].valid := 1, [921].log_data[3].valid := 1, [921].log_data[4].valid := 1, [921].time.Year := 2022, [921].time.Month := 4, [921].time.Day := 27, [921].time.Hour := 2, [921].time.Minute := 19, [921].time.Second := 59, [921].time.DST_ON := 1, [922].log_data[0].min := 1.0, [922].log_data[0].max := 1.0, [922].log_data[0].total := 300.0, [922].log_data[0].time := 300.0, [922].log_data[0].minminute := 20, [922].log_data[0].maxminute := 20, [922].log_data[0].valid := 1, [922].log_data[1].valid := 1, [922].log_data[2].valid := 1, [922].log_data[3].valid := 1, [922].log_data[4].valid := 1, [922].time.Year := 2022, [922].time.Month := 4, [922].time.Day := 27, [922].time.Hour := 2, [922].time.Minute := 24, [922].time.Second := 59, [922].time.DST_ON := 1, [923].log_data[0].min := 1.0, [923].log_data[0].max := 1.0, [923].log_data[0].total := 300.0, [923].log_data[0].time := 300.0, [923].log_data[0].minminute := 25, [923].log_data[0].maxminute := 25, [923].log_data[0].valid := 1, [923].log_data[1].valid := 1, [923].log_data[2].valid := 1, [923].log_data[3].valid := 1, [923].log_data[4].valid := 1, [923].time.Year := 2022, [923].time.Month := 4, [923].time.Day := 27, [923].time.Hour := 2, [923].time.Minute := 29, [923].time.Second := 59, [923].time.DST_ON := 1, [924].log_data[0].min := 1.0, [924].log_data[0].max := 1.0, [924].log_data[0].total := 300.0, [924].log_data[0].time := 300.0, [924].log_data[0].minminute := 30,
        [924].log_data[0].maxminute := 30, [924].log_data[0].valid := 1, [924].log_data[1].valid := 1, [924].log_data[2].valid := 1, [924].log_data[3].valid := 1, [924].log_data[4].valid := 1, [924].time.Year := 2022, [924].time.Month := 4, [924].time.Day := 27, [924].time.Hour := 2, [924].time.Minute := 34, [924].time.Second := 59, [924].time.DST_ON := 1, [925].log_data[0].min := 1.0, [925].log_data[0].max := 1.0, [925].log_data[0].total := 300.0, [925].log_data[0].time := 300.0, [925].log_data[0].minminute := 35, [925].log_data[0].maxminute := 35, [925].log_data[0].valid := 1, [925].log_data[1].valid := 1, [925].log_data[2].valid := 1, [925].log_data[3].valid := 1, [925].log_data[4].valid := 1, [925].time.Year := 2022, [925].time.Month := 4, [925].time.Day := 27, [925].time.Hour := 2, [925].time.Minute := 39, [925].time.Second := 59, [925].time.DST_ON := 1, [926].log_data[0].min := 1.0, [926].log_data[0].max := 1.0, [926].log_data[0].total := 300.0, [926].log_data[0].time := 300.0, [926].log_data[0].minminute := 40, [926].log_data[0].maxminute := 40, [926].log_data[0].valid := 1, [926].log_data[1].valid := 1, [926].log_data[2].valid := 1, [926].log_data[3].valid := 1, [926].log_data[4].valid := 1, [926].time.Year := 2022, [926].time.Month := 4, [926].time.Day := 27, [926].time.Hour := 2, [926].time.Minute := 44, [926].time.Second := 59, [926].time.DST_ON := 1, [927].log_data[0].min := 1.0, [927].log_data[0].max := 1.0, [927].log_data[0].total := 300.0, [927].log_data[0].time := 300.0, [927].log_data[0].minminute := 45, [927].log_data[0].maxminute := 45, [927].log_data[0].valid := 1, [927].log_data[1].valid := 1, [927].log_data[2].valid := 1, [927].log_data[3].valid := 1, [927].log_data[4].valid := 1,
        [927].time.Year := 2022, [927].time.Month := 4, [927].time.Day := 27, [927].time.Hour := 2, [927].time.Minute := 49, [927].time.Second := 59, [927].time.DST_ON := 1, [928].log_data[0].min := 1.0, [928].log_data[0].max := 1.0, [928].log_data[0].total := 300.0, [928].log_data[0].time := 300.0, [928].log_data[0].minminute := 50, [928].log_data[0].maxminute := 50, [928].log_data[0].valid := 1, [928].log_data[1].valid := 1, [928].log_data[2].valid := 1, [928].log_data[3].valid := 1, [928].log_data[4].valid := 1, [928].time.Year := 2022, [928].time.Month := 4, [928].time.Day := 27, [928].time.Hour := 2, [928].time.Minute := 54, [928].time.Second := 59, [928].time.DST_ON := 1, [929].log_data[0].min := 1.0, [929].log_data[0].max := 1.0, [929].log_data[0].total := 300.0, [929].log_data[0].time := 300.0, [929].log_data[0].minminute := 55, [929].log_data[0].maxminute := 55, [929].log_data[0].valid := 1, [929].log_data[1].valid := 1, [929].log_data[2].valid := 1, [929].log_data[3].valid := 1, [929].log_data[4].valid := 1, [929].time.Year := 2022, [929].time.Month := 4, [929].time.Day := 27, [929].time.Hour := 2, [929].time.Minute := 59, [929].time.Second := 59, [929].time.DST_ON := 1, [930].log_data[0].min := 1.0, [930].log_data[0].max := 1.0, [930].log_data[0].total := 299.999, [930].log_data[0].time := 299.999, [930].log_data[0].valid := 1, [930].log_data[1].valid := 1, [930].log_data[2].valid := 1, [930].log_data[3].valid := 1, [930].log_data[4].valid := 1, [930].time.Year := 2022, [930].time.Month := 4, [930].time.Day := 27, [930].time.Hour := 3, [930].time.Minute := 4, [930].time.Second := 59, [930].time.DST_ON := 1, [931].log_data[0].min := 1.0,
        [931].log_data[0].max := 1.0, [931].log_data[0].total := 300.0, [931].log_data[0].time := 300.0, [931].log_data[0].minminute := 5, [931].log_data[0].maxminute := 5, [931].log_data[0].valid := 1, [931].log_data[1].valid := 1, [931].log_data[2].valid := 1, [931].log_data[3].valid := 1, [931].log_data[4].valid := 1, [931].time.Year := 2022, [931].time.Month := 4, [931].time.Day := 27, [931].time.Hour := 3, [931].time.Minute := 9, [931].time.Second := 59, [931].time.DST_ON := 1, [932].log_data[0].min := 1.0, [932].log_data[0].max := 1.0, [932].log_data[0].total := 300.0, [932].log_data[0].time := 300.0, [932].log_data[0].minminute := 10, [932].log_data[0].maxminute := 10, [932].log_data[0].valid := 1, [932].log_data[1].valid := 1, [932].log_data[2].valid := 1, [932].log_data[3].valid := 1, [932].log_data[4].valid := 1, [932].time.Year := 2022, [932].time.Month := 4, [932].time.Day := 27, [932].time.Hour := 3, [932].time.Minute := 14, [932].time.Second := 59, [932].time.DST_ON := 1, [933].log_data[0].min := 1.0, [933].log_data[0].max := 1.0, [933].log_data[0].total := 300.0, [933].log_data[0].time := 300.0, [933].log_data[0].minminute := 15, [933].log_data[0].maxminute := 15, [933].log_data[0].valid := 1, [933].log_data[1].valid := 1, [933].log_data[2].valid := 1, [933].log_data[3].valid := 1, [933].log_data[4].valid := 1, [933].time.Year := 2022, [933].time.Month := 4, [933].time.Day := 27, [933].time.Hour := 3, [933].time.Minute := 19, [933].time.Second := 59, [933].time.DST_ON := 1, [934].log_data[0].min := 1.0, [934].log_data[0].max := 1.0, [934].log_data[0].total := 300.0, [934].log_data[0].time := 300.0, [934].log_data[0].minminute := 20, [934].log_data[0].maxminute := 20, [934].log_data[0].valid := 1,
        [934].log_data[1].valid := 1, [934].log_data[2].valid := 1, [934].log_data[3].valid := 1, [934].log_data[4].valid := 1, [934].time.Year := 2022, [934].time.Month := 4, [934].time.Day := 27, [934].time.Hour := 3, [934].time.Minute := 24, [934].time.Second := 59, [934].time.DST_ON := 1, [935].log_data[0].min := 1.0, [935].log_data[0].max := 1.0, [935].log_data[0].total := 300.0, [935].log_data[0].time := 300.0, [935].log_data[0].minminute := 25, [935].log_data[0].maxminute := 25, [935].log_data[0].valid := 1, [935].log_data[1].valid := 1, [935].log_data[2].valid := 1, [935].log_data[3].valid := 1, [935].log_data[4].valid := 1, [935].time.Year := 2022, [935].time.Month := 4, [935].time.Day := 27, [935].time.Hour := 3, [935].time.Minute := 29, [935].time.Second := 59, [935].time.DST_ON := 1, [936].log_data[0].min := 1.0, [936].log_data[0].max := 1.0, [936].log_data[0].total := 300.0, [936].log_data[0].time := 300.0, [936].log_data[0].minminute := 30, [936].log_data[0].maxminute := 30, [936].log_data[0].valid := 1, [936].log_data[1].valid := 1, [936].log_data[2].valid := 1, [936].log_data[3].valid := 1, [936].log_data[4].valid := 1, [936].time.Year := 2022, [936].time.Month := 4, [936].time.Day := 27, [936].time.Hour := 3, [936].time.Minute := 34, [936].time.Second := 59, [936].time.DST_ON := 1, [937].log_data[0].min := 1.0, [937].log_data[0].max := 1.0, [937].log_data[0].total := 300.0, [937].log_data[0].time := 300.0, [937].log_data[0].minminute := 35, [937].log_data[0].maxminute := 35, [937].log_data[0].valid := 1, [937].log_data[1].valid := 1, [937].log_data[2].valid := 1, [937].log_data[3].valid := 1, [937].log_data[4].valid := 1, [937].time.Year := 2022, [937].time.Month := 4,
        [937].time.Day := 27, [937].time.Hour := 3, [937].time.Minute := 39, [937].time.Second := 59, [937].time.DST_ON := 1, [938].log_data[0].min := 1.0, [938].log_data[0].max := 1.0, [938].log_data[0].total := 300.0, [938].log_data[0].time := 300.0, [938].log_data[0].minminute := 40, [938].log_data[0].maxminute := 40, [938].log_data[0].valid := 1, [938].log_data[1].valid := 1, [938].log_data[2].valid := 1, [938].log_data[3].valid := 1, [938].log_data[4].valid := 1, [938].time.Year := 2022, [938].time.Month := 4, [938].time.Day := 27, [938].time.Hour := 3, [938].time.Minute := 44, [938].time.Second := 59, [938].time.DST_ON := 1, [939].log_data[0].min := 1.0, [939].log_data[0].max := 1.0, [939].log_data[0].total := 300.0, [939].log_data[0].time := 300.0, [939].log_data[0].minminute := 45, [939].log_data[0].maxminute := 45, [939].log_data[0].valid := 1, [939].log_data[1].valid := 1, [939].log_data[2].valid := 1, [939].log_data[3].valid := 1, [939].log_data[4].valid := 1, [939].time.Year := 2022, [939].time.Month := 4, [939].time.Day := 27, [939].time.Hour := 3, [939].time.Minute := 49, [939].time.Second := 59, [939].time.DST_ON := 1, [940].log_data[0].min := 1.0, [940].log_data[0].max := 1.0, [940].log_data[0].total := 300.0, [940].log_data[0].time := 300.0, [940].log_data[0].minminute := 50, [940].log_data[0].maxminute := 50, [940].log_data[0].valid := 1, [940].log_data[1].valid := 1, [940].log_data[2].valid := 1, [940].log_data[3].valid := 1, [940].log_data[4].valid := 1, [940].time.Year := 2022, [940].time.Month := 4, [940].time.Day := 27, [940].time.Hour := 3, [940].time.Minute := 54, [940].time.Second := 59, [940].time.DST_ON := 1, [941].log_data[0].min := 1.0,
        [941].log_data[0].max := 1.0, [941].log_data[0].total := 300.0, [941].log_data[0].time := 300.0, [941].log_data[0].minminute := 55, [941].log_data[0].maxminute := 55, [941].log_data[0].valid := 1, [941].log_data[1].valid := 1, [941].log_data[2].valid := 1, [941].log_data[3].valid := 1, [941].log_data[4].valid := 1, [941].time.Year := 2022, [941].time.Month := 4, [941].time.Day := 27, [941].time.Hour := 3, [941].time.Minute := 59, [941].time.Second := 59, [941].time.DST_ON := 1, [942].log_data[0].min := 1.0, [942].log_data[0].max := 1.0, [942].log_data[0].total := 300.0, [942].log_data[0].time := 300.0, [942].log_data[0].valid := 1, [942].log_data[1].valid := 1, [942].log_data[2].valid := 1, [942].log_data[3].valid := 1, [942].log_data[4].valid := 1, [942].time.Year := 2022, [942].time.Month := 4, [942].time.Day := 27, [942].time.Hour := 4, [942].time.Minute := 4, [942].time.Second := 59, [942].time.DST_ON := 1, [943].log_data[0].min := 1.0, [943].log_data[0].max := 1.0, [943].log_data[0].total := 300.0, [943].log_data[0].time := 300.0, [943].log_data[0].minminute := 5, [943].log_data[0].maxminute := 5, [943].log_data[0].valid := 1, [943].log_data[1].valid := 1, [943].log_data[2].valid := 1, [943].log_data[3].valid := 1, [943].log_data[4].valid := 1, [943].time.Year := 2022, [943].time.Month := 4, [943].time.Day := 27, [943].time.Hour := 4, [943].time.Minute := 9, [943].time.Second := 59, [943].time.DST_ON := 1, [944].log_data[0].min := 1.0, [944].log_data[0].max := 1.0, [944].log_data[0].total := 300.0, [944].log_data[0].time := 300.0, [944].log_data[0].minminute := 10, [944].log_data[0].maxminute := 10, [944].log_data[0].valid := 1, [944].log_data[1].valid := 1, [944].log_data[2].valid := 1,
        [944].log_data[3].valid := 1, [944].log_data[4].valid := 1, [944].time.Year := 2022, [944].time.Month := 4, [944].time.Day := 27, [944].time.Hour := 4, [944].time.Minute := 14, [944].time.Second := 59, [944].time.DST_ON := 1, [945].log_data[0].min := 1.0, [945].log_data[0].max := 1.0, [945].log_data[0].total := 300.0, [945].log_data[0].time := 300.0, [945].log_data[0].minminute := 15, [945].log_data[0].maxminute := 15, [945].log_data[0].valid := 1, [945].log_data[1].valid := 1, [945].log_data[2].valid := 1, [945].log_data[3].valid := 1, [945].log_data[4].valid := 1, [945].time.Year := 2022, [945].time.Month := 4, [945].time.Day := 27, [945].time.Hour := 4, [945].time.Minute := 19, [945].time.Second := 59, [945].time.DST_ON := 1, [946].log_data[0].min := 1.0, [946].log_data[0].max := 1.0, [946].log_data[0].total := 300.0, [946].log_data[0].time := 300.0, [946].log_data[0].minminute := 20, [946].log_data[0].maxminute := 20, [946].log_data[0].valid := 1, [946].log_data[1].valid := 1, [946].log_data[2].valid := 1, [946].log_data[3].valid := 1, [946].log_data[4].valid := 1, [946].time.Year := 2022, [946].time.Month := 4, [946].time.Day := 27, [946].time.Hour := 4, [946].time.Minute := 24, [946].time.Second := 59, [946].time.DST_ON := 1, [947].log_data[0].min := 1.0, [947].log_data[0].max := 1.0, [947].log_data[0].total := 300.0, [947].log_data[0].time := 300.0, [947].log_data[0].minminute := 25, [947].log_data[0].maxminute := 25, [947].log_data[0].valid := 1, [947].log_data[1].valid := 1, [947].log_data[2].valid := 1, [947].log_data[3].valid := 1, [947].log_data[4].valid := 1, [947].time.Year := 2022, [947].time.Month := 4, [947].time.Day := 27, [947].time.Hour := 4,
        [947].time.Minute := 29, [947].time.Second := 59, [947].time.DST_ON := 1, [948].log_data[0].min := 1.0, [948].log_data[0].max := 1.0, [948].log_data[0].total := 300.0, [948].log_data[0].time := 300.0, [948].log_data[0].minminute := 30, [948].log_data[0].maxminute := 30, [948].log_data[0].valid := 1, [948].log_data[1].valid := 1, [948].log_data[2].valid := 1, [948].log_data[3].valid := 1, [948].log_data[4].valid := 1, [948].time.Year := 2022, [948].time.Month := 4, [948].time.Day := 27, [948].time.Hour := 4, [948].time.Minute := 34, [948].time.Second := 59, [948].time.DST_ON := 1, [949].log_data[0].min := 1.0, [949].log_data[0].max := 1.0, [949].log_data[0].total := 300.0, [949].log_data[0].time := 300.0, [949].log_data[0].minminute := 35, [949].log_data[0].maxminute := 35, [949].log_data[0].valid := 1, [949].log_data[1].valid := 1, [949].log_data[2].valid := 1, [949].log_data[3].valid := 1, [949].log_data[4].valid := 1, [949].time.Year := 2022, [949].time.Month := 4, [949].time.Day := 27, [949].time.Hour := 4, [949].time.Minute := 39, [949].time.Second := 59, [949].time.DST_ON := 1, [950].log_data[0].min := 1.0, [950].log_data[0].max := 1.0, [950].log_data[0].total := 300.0, [950].log_data[0].time := 300.0, [950].log_data[0].minminute := 40, [950].log_data[0].maxminute := 40, [950].log_data[0].valid := 1, [950].log_data[1].valid := 1, [950].log_data[2].valid := 1, [950].log_data[3].valid := 1, [950].log_data[4].valid := 1, [950].time.Year := 2022, [950].time.Month := 4, [950].time.Day := 27, [950].time.Hour := 4, [950].time.Minute := 44, [950].time.Second := 59, [950].time.DST_ON := 1, [951].log_data[0].min := 1.0, [951].log_data[0].max := 1.0, [951].log_data[0].total := 300.0,
        [951].log_data[0].time := 300.0, [951].log_data[0].minminute := 45, [951].log_data[0].maxminute := 45, [951].log_data[0].valid := 1, [951].log_data[1].valid := 1, [951].log_data[2].valid := 1, [951].log_data[3].valid := 1, [951].log_data[4].valid := 1, [951].time.Year := 2022, [951].time.Month := 4, [951].time.Day := 27, [951].time.Hour := 4, [951].time.Minute := 49, [951].time.Second := 59, [951].time.DST_ON := 1, [952].log_data[0].min := 1.0, [952].log_data[0].max := 1.0, [952].log_data[0].total := 300.0, [952].log_data[0].time := 300.0, [952].log_data[0].minminute := 50, [952].log_data[0].maxminute := 50, [952].log_data[0].valid := 1, [952].log_data[1].valid := 1, [952].log_data[2].valid := 1, [952].log_data[3].valid := 1, [952].log_data[4].valid := 1, [952].time.Year := 2022, [952].time.Month := 4, [952].time.Day := 27, [952].time.Hour := 4, [952].time.Minute := 54, [952].time.Second := 59, [952].time.DST_ON := 1, [953].log_data[0].min := 1.0, [953].log_data[0].max := 1.0, [953].log_data[0].total := 300.0, [953].log_data[0].time := 300.0, [953].log_data[0].minminute := 55, [953].log_data[0].maxminute := 55, [953].log_data[0].valid := 1, [953].log_data[1].valid := 1, [953].log_data[2].valid := 1, [953].log_data[3].valid := 1, [953].log_data[4].valid := 1, [953].time.Year := 2022, [953].time.Month := 4, [953].time.Day := 27, [953].time.Hour := 4, [953].time.Minute := 59, [953].time.Second := 59, [953].time.DST_ON := 1, [954].log_data[0].min := 1.0, [954].log_data[0].max := 1.0, [954].log_data[0].total := 300.0, [954].log_data[0].time := 300.0, [954].log_data[0].valid := 1, [954].log_data[1].valid := 1, [954].log_data[2].valid := 1, [954].log_data[3].valid := 1, [954].log_data[4].valid := 1,
        [954].time.Year := 2022, [954].time.Month := 4, [954].time.Day := 27, [954].time.Hour := 5, [954].time.Minute := 4, [954].time.Second := 59, [954].time.DST_ON := 1, [955].log_data[0].min := 1.0, [955].log_data[0].max := 1.0, [955].log_data[0].total := 300.0, [955].log_data[0].time := 300.0, [955].log_data[0].minminute := 5, [955].log_data[0].maxminute := 5, [955].log_data[0].valid := 1, [955].log_data[1].valid := 1, [955].log_data[2].valid := 1, [955].log_data[3].valid := 1, [955].log_data[4].valid := 1, [955].time.Year := 2022, [955].time.Month := 4, [955].time.Day := 27, [955].time.Hour := 5, [955].time.Minute := 9, [955].time.Second := 59, [955].time.DST_ON := 1, [956].log_data[0].min := 1.0, [956].log_data[0].max := 1.0, [956].log_data[0].total := 300.0, [956].log_data[0].time := 300.0, [956].log_data[0].minminute := 10, [956].log_data[0].maxminute := 10, [956].log_data[0].valid := 1, [956].log_data[1].valid := 1, [956].log_data[2].valid := 1, [956].log_data[3].valid := 1, [956].log_data[4].valid := 1, [956].time.Year := 2022, [956].time.Month := 4, [956].time.Day := 27, [956].time.Hour := 5, [956].time.Minute := 14, [956].time.Second := 59, [956].time.DST_ON := 1, [957].log_data[0].min := 1.0, [957].log_data[0].max := 1.0, [957].log_data[0].total := 300.0, [957].log_data[0].time := 300.0, [957].log_data[0].minminute := 15, [957].log_data[0].maxminute := 15, [957].log_data[0].valid := 1, [957].log_data[1].valid := 1, [957].log_data[2].valid := 1, [957].log_data[3].valid := 1, [957].log_data[4].valid := 1, [957].time.Year := 2022, [957].time.Month := 4, [957].time.Day := 27, [957].time.Hour := 5, [957].time.Minute := 19, [957].time.Second := 59,
        [957].time.DST_ON := 1, [958].log_data[0].min := 1.0, [958].log_data[0].max := 1.0, [958].log_data[0].total := 300.0, [958].log_data[0].time := 300.0, [958].log_data[0].minminute := 20, [958].log_data[0].maxminute := 20, [958].log_data[0].valid := 1, [958].log_data[1].valid := 1, [958].log_data[2].valid := 1, [958].log_data[3].valid := 1, [958].log_data[4].valid := 1, [958].time.Year := 2022, [958].time.Month := 4, [958].time.Day := 27, [958].time.Hour := 5, [958].time.Minute := 24, [958].time.Second := 59, [958].time.DST_ON := 1, [959].log_data[0].min := 1.0, [959].log_data[0].max := 1.0, [959].log_data[0].total := 300.0, [959].log_data[0].time := 300.0, [959].log_data[0].minminute := 25, [959].log_data[0].maxminute := 25, [959].log_data[0].valid := 1, [959].log_data[1].valid := 1, [959].log_data[2].valid := 1, [959].log_data[3].valid := 1, [959].log_data[4].valid := 1, [959].time.Year := 2022, [959].time.Month := 4, [959].time.Day := 27, [959].time.Hour := 5, [959].time.Minute := 29, [959].time.Second := 59, [959].time.DST_ON := 1, [960].log_data[0].min := 1.0, [960].log_data[0].max := 1.0, [960].log_data[0].total := 299.999, [960].log_data[0].time := 299.999, [960].log_data[0].minminute := 30, [960].log_data[0].maxminute := 30, [960].log_data[0].valid := 1, [960].log_data[1].valid := 1, [960].log_data[2].valid := 1, [960].log_data[3].valid := 1, [960].log_data[4].valid := 1, [960].time.Year := 2022, [960].time.Month := 4, [960].time.Day := 27, [960].time.Hour := 5, [960].time.Minute := 34, [960].time.Second := 59, [960].time.DST_ON := 1, [961].log_data[0].min := 1.0, [961].log_data[0].max := 1.0, [961].log_data[0].total := 300.0, [961].log_data[0].time := 300.0, [961].log_data[0].minminute := 35,
        [961].log_data[0].maxminute := 35, [961].log_data[0].valid := 1, [961].log_data[1].valid := 1, [961].log_data[2].valid := 1, [961].log_data[3].valid := 1, [961].log_data[4].valid := 1, [961].time.Year := 2022, [961].time.Month := 4, [961].time.Day := 27, [961].time.Hour := 5, [961].time.Minute := 39, [961].time.Second := 59, [961].time.DST_ON := 1, [962].log_data[0].min := 1.0, [962].log_data[0].max := 1.0, [962].log_data[0].total := 300.0, [962].log_data[0].time := 300.0, [962].log_data[0].minminute := 40, [962].log_data[0].maxminute := 40, [962].log_data[0].valid := 1, [962].log_data[1].valid := 1, [962].log_data[2].valid := 1, [962].log_data[3].valid := 1, [962].log_data[4].valid := 1, [962].time.Year := 2022, [962].time.Month := 4, [962].time.Day := 27, [962].time.Hour := 5, [962].time.Minute := 44, [962].time.Second := 59, [962].time.DST_ON := 1, [963].log_data[0].min := 1.0, [963].log_data[0].max := 1.0, [963].log_data[0].total := 300.0, [963].log_data[0].time := 300.0, [963].log_data[0].minminute := 45, [963].log_data[0].maxminute := 45, [963].log_data[0].valid := 1, [963].log_data[1].valid := 1, [963].log_data[2].valid := 1, [963].log_data[3].valid := 1, [963].log_data[4].valid := 1, [963].time.Year := 2022, [963].time.Month := 4, [963].time.Day := 27, [963].time.Hour := 5, [963].time.Minute := 49, [963].time.Second := 59, [963].time.DST_ON := 1, [964].log_data[0].min := 1.0, [964].log_data[0].max := 1.0, [964].log_data[0].total := 300.0, [964].log_data[0].time := 300.0, [964].log_data[0].minminute := 50, [964].log_data[0].maxminute := 50, [964].log_data[0].valid := 1, [964].log_data[1].valid := 1, [964].log_data[2].valid := 1, [964].log_data[3].valid := 1, [964].log_data[4].valid := 1,
        [964].time.Year := 2022, [964].time.Month := 4, [964].time.Day := 27, [964].time.Hour := 5, [964].time.Minute := 54, [964].time.Second := 59, [964].time.DST_ON := 1, [965].log_data[0].min := 1.0, [965].log_data[0].max := 1.0, [965].log_data[0].total := 300.0, [965].log_data[0].time := 300.0, [965].log_data[0].minminute := 55, [965].log_data[0].maxminute := 55, [965].log_data[0].valid := 1, [965].log_data[1].valid := 1, [965].log_data[2].valid := 1, [965].log_data[3].valid := 1, [965].log_data[4].valid := 1, [965].time.Year := 2022, [965].time.Month := 4, [965].time.Day := 27, [965].time.Hour := 5, [965].time.Minute := 59, [965].time.Second := 59, [965].time.DST_ON := 1, [966].log_data[0].min := 1.0, [966].log_data[0].max := 1.0, [966].log_data[0].total := 300.0, [966].log_data[0].time := 300.0, [966].log_data[0].valid := 1, [966].log_data[1].valid := 1, [966].log_data[2].valid := 1, [966].log_data[3].valid := 1, [966].log_data[4].valid := 1, [966].time.Year := 2022, [966].time.Month := 4, [966].time.Day := 27, [966].time.Hour := 6, [966].time.Minute := 4, [966].time.Second := 59, [966].time.DST_ON := 1, [967].log_data[0].min := 1.0, [967].log_data[0].max := 1.0, [967].log_data[0].total := 300.0, [967].log_data[0].time := 300.0, [967].log_data[0].minminute := 5, [967].log_data[0].maxminute := 5, [967].log_data[0].valid := 1, [967].log_data[1].valid := 1, [967].log_data[2].valid := 1, [967].log_data[3].valid := 1, [967].log_data[4].valid := 1, [967].time.Year := 2022, [967].time.Month := 4, [967].time.Day := 27, [967].time.Hour := 6, [967].time.Minute := 9, [967].time.Second := 59, [967].time.DST_ON := 1, [968].log_data[0].min := 1.0,
        [968].log_data[0].max := 1.0, [968].log_data[0].total := 300.0, [968].log_data[0].time := 300.0, [968].log_data[0].minminute := 10, [968].log_data[0].maxminute := 10, [968].log_data[0].valid := 1, [968].log_data[1].valid := 1, [968].log_data[2].valid := 1, [968].log_data[3].valid := 1, [968].log_data[4].valid := 1, [968].time.Year := 2022, [968].time.Month := 4, [968].time.Day := 27, [968].time.Hour := 6, [968].time.Minute := 14, [968].time.Second := 59, [968].time.DST_ON := 1, [969].log_data[0].min := 1.0, [969].log_data[0].max := 1.0, [969].log_data[0].total := 300.0, [969].log_data[0].time := 300.0, [969].log_data[0].minminute := 15, [969].log_data[0].maxminute := 15, [969].log_data[0].valid := 1, [969].log_data[1].valid := 1, [969].log_data[2].valid := 1, [969].log_data[3].valid := 1, [969].log_data[4].valid := 1, [969].time.Year := 2022, [969].time.Month := 4, [969].time.Day := 27, [969].time.Hour := 6, [969].time.Minute := 19, [969].time.Second := 59, [969].time.DST_ON := 1, [970].log_data[0].min := 1.0, [970].log_data[0].max := 1.0, [970].log_data[0].total := 300.0, [970].log_data[0].time := 300.0, [970].log_data[0].minminute := 20, [970].log_data[0].maxminute := 20, [970].log_data[0].valid := 1, [970].log_data[1].valid := 1, [970].log_data[2].valid := 1, [970].log_data[3].valid := 1, [970].log_data[4].valid := 1, [970].time.Year := 2022, [970].time.Month := 4, [970].time.Day := 27, [970].time.Hour := 6, [970].time.Minute := 24, [970].time.Second := 59, [970].time.DST_ON := 1, [971].log_data[0].min := 1.0, [971].log_data[0].max := 1.0, [971].log_data[0].total := 300.0, [971].log_data[0].time := 300.0, [971].log_data[0].minminute := 25, [971].log_data[0].maxminute := 25, [971].log_data[0].valid := 1,
        [971].log_data[1].valid := 1, [971].log_data[2].valid := 1, [971].log_data[3].valid := 1, [971].log_data[4].valid := 1, [971].time.Year := 2022, [971].time.Month := 4, [971].time.Day := 27, [971].time.Hour := 6, [971].time.Minute := 29, [971].time.Second := 59, [971].time.DST_ON := 1, [972].log_data[0].min := 1.0, [972].log_data[0].max := 1.0, [972].log_data[0].total := 300.0, [972].log_data[0].time := 300.0, [972].log_data[0].minminute := 30, [972].log_data[0].maxminute := 30, [972].log_data[0].valid := 1, [972].log_data[1].valid := 1, [972].log_data[2].valid := 1, [972].log_data[3].valid := 1, [972].log_data[4].valid := 1, [972].time.Year := 2022, [972].time.Month := 4, [972].time.Day := 27, [972].time.Hour := 6, [972].time.Minute := 34, [972].time.Second := 59, [972].time.DST_ON := 1, [973].log_data[0].min := 1.0, [973].log_data[0].max := 1.0, [973].log_data[0].total := 300.0, [973].log_data[0].time := 300.0, [973].log_data[0].minminute := 35, [973].log_data[0].maxminute := 35, [973].log_data[0].valid := 1, [973].log_data[1].valid := 1, [973].log_data[2].valid := 1, [973].log_data[3].valid := 1, [973].log_data[4].valid := 1, [973].time.Year := 2022, [973].time.Month := 4, [973].time.Day := 27, [973].time.Hour := 6, [973].time.Minute := 39, [973].time.Second := 59, [973].time.DST_ON := 1, [974].log_data[0].min := 1.0, [974].log_data[0].max := 1.0, [974].log_data[0].total := 300.0, [974].log_data[0].time := 300.0, [974].log_data[0].minminute := 40, [974].log_data[0].maxminute := 40, [974].log_data[0].valid := 1, [974].log_data[1].valid := 1, [974].log_data[2].valid := 1, [974].log_data[3].valid := 1, [974].log_data[4].valid := 1, [974].time.Year := 2022, [974].time.Month := 4,
        [974].time.Day := 27, [974].time.Hour := 6, [974].time.Minute := 44, [974].time.Second := 59, [974].time.DST_ON := 1, [975].log_data[0].min := 1.0, [975].log_data[0].max := 1.0, [975].log_data[0].total := 300.0, [975].log_data[0].time := 300.0, [975].log_data[0].minminute := 45, [975].log_data[0].maxminute := 45, [975].log_data[0].valid := 1, [975].log_data[1].valid := 1, [975].log_data[2].valid := 1, [975].log_data[3].valid := 1, [975].log_data[4].valid := 1, [975].time.Year := 2022, [975].time.Month := 4, [975].time.Day := 27, [975].time.Hour := 6, [975].time.Minute := 49, [975].time.Second := 59, [975].time.DST_ON := 1, [976].log_data[0].min := 1.0, [976].log_data[0].max := 1.0, [976].log_data[0].total := 300.0, [976].log_data[0].time := 300.0, [976].log_data[0].minminute := 50, [976].log_data[0].maxminute := 50, [976].log_data[0].valid := 1, [976].log_data[1].valid := 1, [976].log_data[2].valid := 1, [976].log_data[3].valid := 1, [976].log_data[4].valid := 1, [976].time.Year := 2022, [976].time.Month := 4, [976].time.Day := 27, [976].time.Hour := 6, [976].time.Minute := 54, [976].time.Second := 59, [976].time.DST_ON := 1, [977].log_data[0].min := 1.0, [977].log_data[0].max := 1.0, [977].log_data[0].total := 300.0, [977].log_data[0].time := 300.0, [977].log_data[0].minminute := 55, [977].log_data[0].maxminute := 55, [977].log_data[0].valid := 1, [977].log_data[1].valid := 1, [977].log_data[2].valid := 1, [977].log_data[3].valid := 1, [977].log_data[4].valid := 1, [977].time.Year := 2022, [977].time.Month := 4, [977].time.Day := 27, [977].time.Hour := 6, [977].time.Minute := 59, [977].time.Second := 59, [977].time.DST_ON := 1, [978].log_data[0].min := 1.0,
        [978].log_data[0].max := 1.0, [978].log_data[0].total := 300.0, [978].log_data[0].time := 300.0, [978].log_data[0].valid := 1, [978].log_data[1].valid := 1, [978].log_data[2].valid := 1, [978].log_data[3].valid := 1, [978].log_data[4].valid := 1, [978].time.Year := 2022, [978].time.Month := 4, [978].time.Day := 27, [978].time.Hour := 7, [978].time.Minute := 4, [978].time.Second := 59, [978].time.DST_ON := 1, [979].log_data[0].min := 1.0, [979].log_data[0].max := 1.0, [979].log_data[0].total := 300.0, [979].log_data[0].time := 300.0, [979].log_data[0].minminute := 5, [979].log_data[0].maxminute := 5, [979].log_data[0].valid := 1, [979].log_data[1].valid := 1, [979].log_data[2].valid := 1, [979].log_data[3].valid := 1, [979].log_data[4].valid := 1, [979].time.Year := 2022, [979].time.Month := 4, [979].time.Day := 27, [979].time.Hour := 7, [979].time.Minute := 9, [979].time.Second := 59, [979].time.DST_ON := 1, [980].log_data[0].min := 1.0, [980].log_data[0].max := 1.0, [980].log_data[0].total := 300.0, [980].log_data[0].time := 300.0, [980].log_data[0].minminute := 10, [980].log_data[0].maxminute := 10, [980].log_data[0].valid := 1, [980].log_data[1].valid := 1, [980].log_data[2].valid := 1, [980].log_data[3].valid := 1, [980].log_data[4].valid := 1, [980].time.Year := 2022, [980].time.Month := 4, [980].time.Day := 27, [980].time.Hour := 7, [980].time.Minute := 14, [980].time.Second := 59, [980].time.DST_ON := 1, [981].log_data[0].min := 1.0, [981].log_data[0].max := 1.0, [981].log_data[0].total := 300.0, [981].log_data[0].time := 300.0, [981].log_data[0].minminute := 15, [981].log_data[0].maxminute := 15, [981].log_data[0].valid := 1, [981].log_data[1].valid := 1, [981].log_data[2].valid := 1,
        [981].log_data[3].valid := 1, [981].log_data[4].valid := 1, [981].time.Year := 2022, [981].time.Month := 4, [981].time.Day := 27, [981].time.Hour := 7, [981].time.Minute := 19, [981].time.Second := 59, [981].time.DST_ON := 1, [982].log_data[0].min := 1.0, [982].log_data[0].max := 1.0, [982].log_data[0].total := 300.0, [982].log_data[0].time := 300.0, [982].log_data[0].minminute := 20, [982].log_data[0].maxminute := 20, [982].log_data[0].valid := 1, [982].log_data[1].valid := 1, [982].log_data[2].valid := 1, [982].log_data[3].valid := 1, [982].log_data[4].valid := 1, [982].time.Year := 2022, [982].time.Month := 4, [982].time.Day := 27, [982].time.Hour := 7, [982].time.Minute := 24, [982].time.Second := 59, [982].time.DST_ON := 1, [983].log_data[0].min := 1.0, [983].log_data[0].max := 1.0, [983].log_data[0].total := 300.0, [983].log_data[0].time := 300.0, [983].log_data[0].minminute := 25, [983].log_data[0].maxminute := 25, [983].log_data[0].valid := 1, [983].log_data[1].valid := 1, [983].log_data[2].valid := 1, [983].log_data[3].valid := 1, [983].log_data[4].valid := 1, [983].time.Year := 2022, [983].time.Month := 4, [983].time.Day := 27, [983].time.Hour := 7, [983].time.Minute := 29, [983].time.Second := 59, [983].time.DST_ON := 1, [984].log_data[0].min := 1.0, [984].log_data[0].max := 1.0, [984].log_data[0].total := 300.0, [984].log_data[0].time := 300.0, [984].log_data[0].minminute := 30, [984].log_data[0].maxminute := 30, [984].log_data[0].valid := 1, [984].log_data[1].valid := 1, [984].log_data[2].valid := 1, [984].log_data[3].valid := 1, [984].log_data[4].valid := 1, [984].time.Year := 2022, [984].time.Month := 4, [984].time.Day := 27, [984].time.Hour := 7,
        [984].time.Minute := 34, [984].time.Second := 59, [984].time.DST_ON := 1, [985].log_data[0].min := 1.0, [985].log_data[0].max := 1.0, [985].log_data[0].total := 300.0, [985].log_data[0].time := 300.0, [985].log_data[0].minminute := 35, [985].log_data[0].maxminute := 35, [985].log_data[0].valid := 1, [985].log_data[1].valid := 1, [985].log_data[2].valid := 1, [985].log_data[3].valid := 1, [985].log_data[4].valid := 1, [985].time.Year := 2022, [985].time.Month := 4, [985].time.Day := 27, [985].time.Hour := 7, [985].time.Minute := 39, [985].time.Second := 59, [985].time.DST_ON := 1, [986].log_data[0].min := 1.0, [986].log_data[0].max := 1.0, [986].log_data[0].total := 300.0, [986].log_data[0].time := 300.0, [986].log_data[0].minminute := 40, [986].log_data[0].maxminute := 40, [986].log_data[0].valid := 1, [986].log_data[1].valid := 1, [986].log_data[2].valid := 1, [986].log_data[3].valid := 1, [986].log_data[4].valid := 1, [986].time.Year := 2022, [986].time.Month := 4, [986].time.Day := 27, [986].time.Hour := 7, [986].time.Minute := 44, [986].time.Second := 59, [986].time.DST_ON := 1, [987].log_data[0].min := 1.0, [987].log_data[0].max := 1.0, [987].log_data[0].total := 300.0, [987].log_data[0].time := 300.0, [987].log_data[0].minminute := 45, [987].log_data[0].maxminute := 45, [987].log_data[0].valid := 1, [987].log_data[1].valid := 1, [987].log_data[2].valid := 1, [987].log_data[3].valid := 1, [987].log_data[4].valid := 1, [987].time.Year := 2022, [987].time.Month := 4, [987].time.Day := 27, [987].time.Hour := 7, [987].time.Minute := 49, [987].time.Second := 59, [987].time.DST_ON := 1, [988].log_data[0].min := 1.0, [988].log_data[0].max := 1.0, [988].log_data[0].total := 300.0,
        [988].log_data[0].time := 300.0, [988].log_data[0].minminute := 50, [988].log_data[0].maxminute := 50, [988].log_data[0].valid := 1, [988].log_data[1].valid := 1, [988].log_data[2].valid := 1, [988].log_data[3].valid := 1, [988].log_data[4].valid := 1, [988].time.Year := 2022, [988].time.Month := 4, [988].time.Day := 27, [988].time.Hour := 7, [988].time.Minute := 54, [988].time.Second := 59, [988].time.DST_ON := 1, [989].log_data[0].min := 1.0, [989].log_data[0].max := 1.0, [989].log_data[0].total := 300.0, [989].log_data[0].time := 300.0, [989].log_data[0].minminute := 55, [989].log_data[0].maxminute := 55, [989].log_data[0].valid := 1, [989].log_data[1].valid := 1, [989].log_data[2].valid := 1, [989].log_data[3].valid := 1, [989].log_data[4].valid := 1, [989].time.Year := 2022, [989].time.Month := 4, [989].time.Day := 27, [989].time.Hour := 7, [989].time.Minute := 59, [989].time.Second := 59, [989].time.DST_ON := 1, [990].log_data[0].min := 1.0, [990].log_data[0].max := 1.0, [990].log_data[0].total := 300.0, [990].log_data[0].time := 300.0, [990].log_data[0].valid := 1, [990].log_data[1].valid := 1, [990].log_data[2].valid := 1, [990].log_data[3].valid := 1, [990].log_data[4].valid := 1, [990].time.Year := 2022, [990].time.Month := 4, [990].time.Day := 27, [990].time.Hour := 8, [990].time.Minute := 4, [990].time.Second := 59, [990].time.DST_ON := 1, [991].log_data[0].min := 1.0, [991].log_data[0].max := 1.0, [991].log_data[0].total := 300.0, [991].log_data[0].time := 300.0, [991].log_data[0].minminute := 5, [991].log_data[0].maxminute := 5, [991].log_data[0].valid := 1, [991].log_data[1].valid := 1, [991].log_data[2].valid := 1, [991].log_data[3].valid := 1, [991].log_data[4].valid := 1,
        [991].time.Year := 2022, [991].time.Month := 4, [991].time.Day := 27, [991].time.Hour := 8, [991].time.Minute := 9, [991].time.Second := 59, [991].time.DST_ON := 1, [992].log_data[0].min := 1.0, [992].log_data[0].max := 1.0, [992].log_data[0].total := 300.0, [992].log_data[0].time := 300.0, [992].log_data[0].minminute := 10, [992].log_data[0].maxminute := 10, [992].log_data[0].valid := 1, [992].log_data[1].valid := 1, [992].log_data[2].valid := 1, [992].log_data[3].valid := 1, [992].log_data[4].valid := 1, [992].time.Year := 2022, [992].time.Month := 4, [992].time.Day := 27, [992].time.Hour := 8, [992].time.Minute := 14, [992].time.Second := 59, [992].time.DST_ON := 1, [993].log_data[0].min := 1.0, [993].log_data[0].max := 1.0, [993].log_data[0].total := 300.0, [993].log_data[0].time := 300.0, [993].log_data[0].minminute := 15, [993].log_data[0].maxminute := 15, [993].log_data[0].valid := 1, [993].log_data[1].valid := 1, [993].log_data[2].valid := 1, [993].log_data[3].valid := 1, [993].log_data[4].valid := 1, [993].time.Year := 2022, [993].time.Month := 4, [993].time.Day := 27, [993].time.Hour := 8, [993].time.Minute := 19, [993].time.Second := 59, [993].time.DST_ON := 1, [994].log_data[0].min := 1.0, [994].log_data[0].max := 1.0, [994].log_data[0].total := 300.0, [994].log_data[0].time := 300.0, [994].log_data[0].minminute := 20, [994].log_data[0].maxminute := 20, [994].log_data[0].valid := 1, [994].log_data[1].valid := 1, [994].log_data[2].valid := 1, [994].log_data[3].valid := 1, [994].log_data[4].valid := 1, [994].time.Year := 2022, [994].time.Month := 4, [994].time.Day := 27, [994].time.Hour := 8, [994].time.Minute := 24, [994].time.Second := 59,
        [994].time.DST_ON := 1, [995].log_data[0].min := 1.0, [995].log_data[0].max := 1.0, [995].log_data[0].total := 300.0, [995].log_data[0].time := 300.0, [995].log_data[0].minminute := 25, [995].log_data[0].maxminute := 25, [995].log_data[0].valid := 1, [995].log_data[1].valid := 1, [995].log_data[2].valid := 1, [995].log_data[3].valid := 1, [995].log_data[4].valid := 1, [995].time.Year := 2022, [995].time.Month := 4, [995].time.Day := 27, [995].time.Hour := 8, [995].time.Minute := 29, [995].time.Second := 59, [995].time.DST_ON := 1, [996].log_data[0].min := 1.0, [996].log_data[0].max := 1.0, [996].log_data[0].total := 300.0, [996].log_data[0].time := 300.0, [996].log_data[0].minminute := 30, [996].log_data[0].maxminute := 30, [996].log_data[0].valid := 1, [996].log_data[1].valid := 1, [996].log_data[2].valid := 1, [996].log_data[3].valid := 1, [996].log_data[4].valid := 1, [996].time.Year := 2022, [996].time.Month := 4, [996].time.Day := 27, [996].time.Hour := 8, [996].time.Minute := 34, [996].time.Second := 59, [996].time.DST_ON := 1, [997].log_data[0].min := 1.0, [997].log_data[0].max := 1.0, [997].log_data[0].total := 300.0, [997].log_data[0].time := 300.0, [997].log_data[0].minminute := 35, [997].log_data[0].maxminute := 35, [997].log_data[0].valid := 1, [997].log_data[1].valid := 1, [997].log_data[2].valid := 1, [997].log_data[3].valid := 1, [997].log_data[4].valid := 1, [997].time.Year := 2022, [997].time.Month := 4, [997].time.Day := 27, [997].time.Hour := 8, [997].time.Minute := 39, [997].time.Second := 59, [997].time.DST_ON := 1, [998].log_data[0].min := 1.0, [998].log_data[0].max := 1.0, [998].log_data[0].total := 300.0, [998].log_data[0].time := 300.0, [998].log_data[0].minminute := 40,
        [998].log_data[0].maxminute := 40, [998].log_data[0].valid := 1, [998].log_data[1].valid := 1, [998].log_data[2].valid := 1, [998].log_data[3].valid := 1, [998].log_data[4].valid := 1, [998].time.Year := 2022, [998].time.Month := 4, [998].time.Day := 27, [998].time.Hour := 8, [998].time.Minute := 44, [998].time.Second := 59, [998].time.DST_ON := 1, [999].log_data[0].min := 1.0, [999].log_data[0].max := 1.0, [999].log_data[0].total := 300.0, [999].log_data[0].time := 300.0, [999].log_data[0].minminute := 45, [999].log_data[0].maxminute := 45, [999].log_data[0].valid := 1, [999].log_data[1].valid := 1, [999].log_data[2].valid := 1, [999].log_data[3].valid := 1, [999].log_data[4].valid := 1, [999].time.Year := 2022, [999].time.Month := 4, [999].time.Day := 27, [999].time.Hour := 8, [999].time.Minute := 49, [999].time.Second := 59, [999].time.DST_ON := 1, [1000].log_data[0].min := 1.0, [1000].log_data[0].max := 1.0, [1000].log_data[0].total := 300.0, [1000].log_data[0].time := 300.0, [1000].log_data[0].minminute := 50, [1000].log_data[0].maxminute := 50, [1000].log_data[0].valid := 1, [1000].log_data[1].valid := 1, [1000].log_data[2].valid := 1, [1000].log_data[3].valid := 1, [1000].log_data[4].valid := 1, [1000].time.Year := 2022, [1000].time.Month := 4, [1000].time.Day := 27, [1000].time.Hour := 8, [1000].time.Minute := 54, [1000].time.Second := 59, [1000].time.DST_ON := 1, [1001].log_data[0].min := 1.0, [1001].log_data[0].max := 1.0, [1001].log_data[0].total := 300.0, [1001].log_data[0].time := 300.0, [1001].log_data[0].minminute := 55, [1001].log_data[0].maxminute := 55, [1001].log_data[0].valid := 1, [1001].log_data[1].valid := 1, [1001].log_data[2].valid := 1, [1001].log_data[3].valid := 1, [1001].log_data[4].valid := 1,
        [1001].time.Year := 2022, [1001].time.Month := 4, [1001].time.Day := 27, [1001].time.Hour := 8, [1001].time.Minute := 59, [1001].time.Second := 59, [1001].time.DST_ON := 1, [1002].log_data[0].min := 1.0, [1002].log_data[0].max := 1.0, [1002].log_data[0].total := 300.0, [1002].log_data[0].time := 300.0, [1002].log_data[0].valid := 1, [1002].log_data[1].valid := 1, [1002].log_data[2].valid := 1, [1002].log_data[3].valid := 1, [1002].log_data[4].valid := 1, [1002].time.Year := 2022, [1002].time.Month := 4, [1002].time.Day := 27, [1002].time.Hour := 9, [1002].time.Minute := 4, [1002].time.Second := 59, [1002].time.DST_ON := 1, [1003].log_data[0].min := 1.0, [1003].log_data[0].max := 1.0, [1003].log_data[0].total := 300.0, [1003].log_data[0].time := 300.0, [1003].log_data[0].minminute := 5, [1003].log_data[0].maxminute := 5, [1003].log_data[0].valid := 1, [1003].log_data[1].valid := 1, [1003].log_data[2].valid := 1, [1003].log_data[3].valid := 1, [1003].log_data[4].valid := 1, [1003].time.Year := 2022, [1003].time.Month := 4, [1003].time.Day := 27, [1003].time.Hour := 9, [1003].time.Minute := 9, [1003].time.Second := 59, [1003].time.DST_ON := 1, [1004].log_data[0].min := 1.0, [1004].log_data[0].max := 1.0, [1004].log_data[0].total := 300.0, [1004].log_data[0].time := 300.0, [1004].log_data[0].minminute := 10, [1004].log_data[0].maxminute := 10, [1004].log_data[0].valid := 1, [1004].log_data[1].valid := 1, [1004].log_data[2].valid := 1, [1004].log_data[3].valid := 1, [1004].log_data[4].valid := 1, [1004].time.Year := 2022, [1004].time.Month := 4, [1004].time.Day := 27, [1004].time.Hour := 9, [1004].time.Minute := 14, [1004].time.Second := 59, [1004].time.DST_ON := 1, [1005].log_data[0].min := 1.0,
        [1005].log_data[0].max := 1.0, [1005].log_data[0].total := 300.0, [1005].log_data[0].time := 300.0, [1005].log_data[0].minminute := 15, [1005].log_data[0].maxminute := 15, [1005].log_data[0].valid := 1, [1005].log_data[1].valid := 1, [1005].log_data[2].valid := 1, [1005].log_data[3].valid := 1, [1005].log_data[4].valid := 1, [1005].time.Year := 2022, [1005].time.Month := 4, [1005].time.Day := 27, [1005].time.Hour := 9, [1005].time.Minute := 19, [1005].time.Second := 59, [1005].time.DST_ON := 1, [1006].log_data[0].min := 1.0, [1006].log_data[0].max := 1.0, [1006].log_data[0].total := 300.0, [1006].log_data[0].time := 300.0, [1006].log_data[0].minminute := 20, [1006].log_data[0].maxminute := 20, [1006].log_data[0].valid := 1, [1006].log_data[1].valid := 1, [1006].log_data[2].valid := 1, [1006].log_data[3].valid := 1, [1006].log_data[4].valid := 1, [1006].time.Year := 2022, [1006].time.Month := 4, [1006].time.Day := 27, [1006].time.Hour := 9, [1006].time.Minute := 24, [1006].time.Second := 59, [1006].time.DST_ON := 1, [1007].log_data[0].min := 1.0, [1007].log_data[0].max := 1.0, [1007].log_data[0].total := 300.0, [1007].log_data[0].time := 300.0, [1007].log_data[0].minminute := 25, [1007].log_data[0].maxminute := 25, [1007].log_data[0].valid := 1, [1007].log_data[1].valid := 1, [1007].log_data[2].valid := 1, [1007].log_data[3].valid := 1, [1007].log_data[4].valid := 1, [1007].time.Year := 2022, [1007].time.Month := 4, [1007].time.Day := 27, [1007].time.Hour := 9, [1007].time.Minute := 29, [1007].time.Second := 59, [1007].time.DST_ON := 1, [1008].log_data[0].min := 1.0, [1008].log_data[0].max := 1.0, [1008].log_data[0].total := 300.0, [1008].log_data[0].time := 300.0, [1008].log_data[0].minminute := 30, [1008].log_data[0].maxminute := 30, [1008].log_data[0].valid := 1,
        [1008].log_data[1].valid := 1, [1008].log_data[2].valid := 1, [1008].log_data[3].valid := 1, [1008].log_data[4].valid := 1, [1008].time.Year := 2022, [1008].time.Month := 4, [1008].time.Day := 27, [1008].time.Hour := 9, [1008].time.Minute := 34, [1008].time.Second := 59, [1008].time.DST_ON := 1, [1009].log_data[0].min := 1.0, [1009].log_data[0].max := 1.0, [1009].log_data[0].total := 300.0, [1009].log_data[0].time := 300.0, [1009].log_data[0].minminute := 35, [1009].log_data[0].maxminute := 35, [1009].log_data[0].valid := 1, [1009].log_data[1].valid := 1, [1009].log_data[2].valid := 1, [1009].log_data[3].valid := 1, [1009].log_data[4].valid := 1, [1009].time.Year := 2022, [1009].time.Month := 4, [1009].time.Day := 27, [1009].time.Hour := 9, [1009].time.Minute := 39, [1009].time.Second := 59, [1009].time.DST_ON := 1, [1010].log_data[0].min := 1.0, [1010].log_data[0].max := 1.0, [1010].log_data[0].total := 300.0, [1010].log_data[0].time := 300.0, [1010].log_data[0].minminute := 40, [1010].log_data[0].maxminute := 40, [1010].log_data[0].valid := 1, [1010].log_data[1].valid := 1, [1010].log_data[2].valid := 1, [1010].log_data[3].valid := 1, [1010].log_data[4].valid := 1, [1010].time.Year := 2022, [1010].time.Month := 4, [1010].time.Day := 27, [1010].time.Hour := 9, [1010].time.Minute := 44, [1010].time.Second := 59, [1010].time.DST_ON := 1, [1011].log_data[0].min := 1.0, [1011].log_data[0].max := 1.0, [1011].log_data[0].total := 300.0, [1011].log_data[0].time := 300.0, [1011].log_data[0].minminute := 45, [1011].log_data[0].maxminute := 45, [1011].log_data[0].valid := 1, [1011].log_data[1].valid := 1, [1011].log_data[2].valid := 1, [1011].log_data[3].valid := 1, [1011].log_data[4].valid := 1, [1011].time.Year := 2022, [1011].time.Month := 4,
        [1011].time.Day := 27, [1011].time.Hour := 9, [1011].time.Minute := 49, [1011].time.Second := 59, [1011].time.DST_ON := 1, [1012].log_data[0].min := 1.0, [1012].log_data[0].max := 1.0, [1012].log_data[0].total := 300.0, [1012].log_data[0].time := 300.0, [1012].log_data[0].minminute := 50, [1012].log_data[0].maxminute := 50, [1012].log_data[0].valid := 1, [1012].log_data[1].valid := 1, [1012].log_data[2].valid := 1, [1012].log_data[3].valid := 1, [1012].log_data[4].valid := 1, [1012].time.Year := 2022, [1012].time.Month := 4, [1012].time.Day := 27, [1012].time.Hour := 9, [1012].time.Minute := 54, [1012].time.Second := 59, [1012].time.DST_ON := 1, [1013].log_data[0].min := 1.0, [1013].log_data[0].max := 1.0, [1013].log_data[0].total := 300.0, [1013].log_data[0].time := 300.0, [1013].log_data[0].minminute := 55, [1013].log_data[0].maxminute := 55, [1013].log_data[0].valid := 1, [1013].log_data[1].valid := 1, [1013].log_data[2].valid := 1, [1013].log_data[3].valid := 1, [1013].log_data[4].valid := 1, [1013].time.Year := 2022, [1013].time.Month := 4, [1013].time.Day := 27, [1013].time.Hour := 9, [1013].time.Minute := 59, [1013].time.Second := 59, [1013].time.DST_ON := 1, [1014].log_data[0].min := 1.0, [1014].log_data[0].max := 1.0, [1014].log_data[0].total := 300.0, [1014].log_data[0].time := 300.0, [1014].log_data[0].valid := 1, [1014].log_data[1].valid := 1, [1014].log_data[2].valid := 1, [1014].log_data[3].valid := 1, [1014].log_data[4].valid := 1, [1014].time.Year := 2022, [1014].time.Month := 4, [1014].time.Day := 27, [1014].time.Hour := 10, [1014].time.Minute := 4, [1014].time.Second := 59, [1014].time.DST_ON := 1, [1015].log_data[0].min := 1.0, [1015].log_data[0].max := 1.0, [1015].log_data[0].total := 300.0,
        [1015].log_data[0].time := 300.0, [1015].log_data[0].minminute := 5, [1015].log_data[0].maxminute := 5, [1015].log_data[0].valid := 1, [1015].log_data[1].valid := 1, [1015].log_data[2].valid := 1, [1015].log_data[3].valid := 1, [1015].log_data[4].valid := 1, [1015].time.Year := 2022, [1015].time.Month := 4, [1015].time.Day := 27, [1015].time.Hour := 10, [1015].time.Minute := 9, [1015].time.Second := 59, [1015].time.DST_ON := 1, [1016].log_data[0].min := 1.0, [1016].log_data[0].max := 1.0, [1016].log_data[0].total := 300.0, [1016].log_data[0].time := 300.0, [1016].log_data[0].minminute := 10, [1016].log_data[0].maxminute := 10, [1016].log_data[0].valid := 1, [1016].log_data[1].valid := 1, [1016].log_data[2].valid := 1, [1016].log_data[3].valid := 1, [1016].log_data[4].valid := 1, [1016].time.Year := 2022, [1016].time.Month := 4, [1016].time.Day := 27, [1016].time.Hour := 10, [1016].time.Minute := 14, [1016].time.Second := 59, [1016].time.DST_ON := 1, [1017].log_data[0].min := 1.0, [1017].log_data[0].max := 1.0, [1017].log_data[0].total := 300.0, [1017].log_data[0].time := 300.0, [1017].log_data[0].minminute := 15, [1017].log_data[0].maxminute := 15, [1017].log_data[0].valid := 1, [1017].log_data[1].valid := 1, [1017].log_data[2].valid := 1, [1017].log_data[3].valid := 1, [1017].log_data[4].valid := 1, [1017].time.Year := 2022, [1017].time.Month := 4, [1017].time.Day := 27, [1017].time.Hour := 10, [1017].time.Minute := 19, [1017].time.Second := 59, [1017].time.DST_ON := 1, [1018].log_data[0].min := 1.0, [1018].log_data[0].max := 1.0, [1018].log_data[0].total := 300.0, [1018].log_data[0].time := 300.0, [1018].log_data[0].minminute := 20, [1018].log_data[0].maxminute := 20, [1018].log_data[0].valid := 1, [1018].log_data[1].valid := 1, [1018].log_data[2].valid := 1,
        [1018].log_data[3].valid := 1, [1018].log_data[4].valid := 1, [1018].time.Year := 2022, [1018].time.Month := 4, [1018].time.Day := 27, [1018].time.Hour := 10, [1018].time.Minute := 24, [1018].time.Second := 59, [1018].time.DST_ON := 1, [1019].log_data[0].min := 1.0, [1019].log_data[0].max := 1.0, [1019].log_data[0].total := 300.0, [1019].log_data[0].time := 300.0, [1019].log_data[0].minminute := 25, [1019].log_data[0].maxminute := 25, [1019].log_data[0].valid := 1, [1019].log_data[1].valid := 1, [1019].log_data[2].valid := 1, [1019].log_data[3].valid := 1, [1019].log_data[4].valid := 1, [1019].time.Year := 2022, [1019].time.Month := 4, [1019].time.Day := 27, [1019].time.Hour := 10, [1019].time.Minute := 29, [1019].time.Second := 59, [1019].time.DST_ON := 1, [1020].log_data[0].min := 1.0, [1020].log_data[0].max := 1.0, [1020].log_data[0].total := 300.0, [1020].log_data[0].time := 300.0, [1020].log_data[0].minminute := 30, [1020].log_data[0].maxminute := 30, [1020].log_data[0].valid := 1, [1020].log_data[1].valid := 1, [1020].log_data[2].valid := 1, [1020].log_data[3].valid := 1, [1020].log_data[4].valid := 1, [1020].time.Year := 2022, [1020].time.Month := 4, [1020].time.Day := 27, [1020].time.Hour := 10, [1020].time.Minute := 34, [1020].time.Second := 59, [1020].time.DST_ON := 1, [1021].log_data[0].min := 1.0, [1021].log_data[0].max := 1.0, [1021].log_data[0].total := 300.0, [1021].log_data[0].time := 300.0, [1021].log_data[0].minminute := 35, [1021].log_data[0].maxminute := 35, [1021].log_data[0].valid := 1, [1021].log_data[1].valid := 1, [1021].log_data[2].valid := 1, [1021].log_data[3].valid := 1, [1021].log_data[4].valid := 1, [1021].time.Year := 2022, [1021].time.Month := 4, [1021].time.Day := 27, [1021].time.Hour := 10,
        [1021].time.Minute := 39, [1021].time.Second := 59, [1021].time.DST_ON := 1, [1022].log_data[0].min := 1.0, [1022].log_data[0].max := 1.0, [1022].log_data[0].total := 300.0, [1022].log_data[0].time := 300.0, [1022].log_data[0].minminute := 40, [1022].log_data[0].maxminute := 40, [1022].log_data[0].valid := 1, [1022].log_data[1].valid := 1, [1022].log_data[2].valid := 1, [1022].log_data[3].valid := 1, [1022].log_data[4].valid := 1, [1022].time.Year := 2022, [1022].time.Month := 4, [1022].time.Day := 27, [1022].time.Hour := 10, [1022].time.Minute := 44, [1022].time.Second := 59, [1022].time.DST_ON := 1, [1023].log_data[0].min := 1.0, [1023].log_data[0].max := 1.0, [1023].log_data[0].total := 300.0, [1023].log_data[0].time := 300.0, [1023].log_data[0].minminute := 45, [1023].log_data[0].maxminute := 45, [1023].log_data[0].valid := 1, [1023].log_data[1].valid := 1, [1023].log_data[2].valid := 1, [1023].log_data[3].valid := 1, [1023].log_data[4].valid := 1, [1023].time.Year := 2022, [1023].time.Month := 4, [1023].time.Day := 27, [1023].time.Hour := 10, [1023].time.Minute := 49, [1023].time.Second := 59, [1023].time.DST_ON := 1, [1024].log_data[0].min := 1.0, [1024].log_data[0].max := 1.0, [1024].log_data[0].total := 300.0, [1024].log_data[0].time := 300.0, [1024].log_data[0].minminute := 50, [1024].log_data[0].maxminute := 50, [1024].log_data[0].valid := 1, [1024].log_data[1].valid := 1, [1024].log_data[2].valid := 1, [1024].log_data[3].valid := 1, [1024].log_data[4].valid := 1, [1024].time.Year := 2022, [1024].time.Month := 4, [1024].time.Day := 27, [1024].time.Hour := 10, [1024].time.Minute := 54, [1024].time.Second := 59, [1024].time.DST_ON := 1, [1025].log_data[0].min := 1.0, [1025].log_data[0].max := 1.0, [1025].log_data[0].total := 300.0,
        [1025].log_data[0].time := 300.0, [1025].log_data[0].minminute := 55, [1025].log_data[0].maxminute := 55, [1025].log_data[0].valid := 1, [1025].log_data[1].valid := 1, [1025].log_data[2].valid := 1, [1025].log_data[3].valid := 1, [1025].log_data[4].valid := 1, [1025].time.Year := 2022, [1025].time.Month := 4, [1025].time.Day := 27, [1025].time.Hour := 10, [1025].time.Minute := 59, [1025].time.Second := 59, [1025].time.DST_ON := 1, [1026].log_data[0].min := 1.0, [1026].log_data[0].max := 1.0, [1026].log_data[0].total := 300.0, [1026].log_data[0].time := 300.0, [1026].log_data[0].valid := 1, [1026].log_data[1].valid := 1, [1026].log_data[2].valid := 1, [1026].log_data[3].valid := 1, [1026].log_data[4].valid := 1, [1026].time.Year := 2022, [1026].time.Month := 4, [1026].time.Day := 27, [1026].time.Hour := 11, [1026].time.Minute := 4, [1026].time.Second := 59, [1026].time.DST_ON := 1, [1027].log_data[0].min := 1.0, [1027].log_data[0].max := 1.0, [1027].log_data[0].total := 300.0, [1027].log_data[0].time := 300.0, [1027].log_data[0].minminute := 5, [1027].log_data[0].maxminute := 5, [1027].log_data[0].valid := 1, [1027].log_data[1].valid := 1, [1027].log_data[2].valid := 1, [1027].log_data[3].valid := 1, [1027].log_data[4].valid := 1, [1027].time.Year := 2022, [1027].time.Month := 4, [1027].time.Day := 27, [1027].time.Hour := 11, [1027].time.Minute := 9, [1027].time.Second := 59, [1027].time.DST_ON := 1, [1028].log_data[0].min := 1.0, [1028].log_data[0].max := 1.0, [1028].log_data[0].total := 300.0, [1028].log_data[0].time := 300.0, [1028].log_data[0].minminute := 10, [1028].log_data[0].maxminute := 10, [1028].log_data[0].valid := 1, [1028].log_data[1].valid := 1, [1028].log_data[2].valid := 1, [1028].log_data[3].valid := 1, [1028].log_data[4].valid := 1,
        [1028].time.Year := 2022, [1028].time.Month := 4, [1028].time.Day := 27, [1028].time.Hour := 11, [1028].time.Minute := 14, [1028].time.Second := 59, [1028].time.DST_ON := 1, [1029].log_data[0].min := 1.0, [1029].log_data[0].max := 1.0, [1029].log_data[0].total := 300.0, [1029].log_data[0].time := 300.0, [1029].log_data[0].minminute := 15, [1029].log_data[0].maxminute := 15, [1029].log_data[0].valid := 1, [1029].log_data[1].valid := 1, [1029].log_data[2].valid := 1, [1029].log_data[3].valid := 1, [1029].log_data[4].valid := 1, [1029].time.Year := 2022, [1029].time.Month := 4, [1029].time.Day := 27, [1029].time.Hour := 11, [1029].time.Minute := 19, [1029].time.Second := 59, [1029].time.DST_ON := 1, [1030].log_data[0].min := 1.0, [1030].log_data[0].max := 1.0, [1030].log_data[0].total := 300.0, [1030].log_data[0].time := 300.0, [1030].log_data[0].minminute := 20, [1030].log_data[0].maxminute := 20, [1030].log_data[0].valid := 1, [1030].log_data[1].valid := 1, [1030].log_data[2].valid := 1, [1030].log_data[3].valid := 1, [1030].log_data[4].valid := 1, [1030].time.Year := 2022, [1030].time.Month := 4, [1030].time.Day := 27, [1030].time.Hour := 11, [1030].time.Minute := 24, [1030].time.Second := 59, [1030].time.DST_ON := 1, [1031].log_data[0].min := 1.0, [1031].log_data[0].max := 1.0, [1031].log_data[0].total := 300.0, [1031].log_data[0].time := 300.0, [1031].log_data[0].minminute := 25, [1031].log_data[0].maxminute := 25, [1031].log_data[0].valid := 1, [1031].log_data[1].valid := 1, [1031].log_data[2].valid := 1, [1031].log_data[3].valid := 1, [1031].log_data[4].valid := 1, [1031].time.Year := 2022, [1031].time.Month := 4, [1031].time.Day := 27, [1031].time.Hour := 11, [1031].time.Minute := 29, [1031].time.Second := 59,
        [1031].time.DST_ON := 1, [1032].log_data[0].min := 1.0, [1032].log_data[0].max := 1.0, [1032].log_data[0].total := 300.0, [1032].log_data[0].time := 300.0, [1032].log_data[0].minminute := 30, [1032].log_data[0].maxminute := 30, [1032].log_data[0].valid := 1, [1032].log_data[1].valid := 1, [1032].log_data[2].valid := 1, [1032].log_data[3].valid := 1, [1032].log_data[4].valid := 1, [1032].time.Year := 2022, [1032].time.Month := 4, [1032].time.Day := 27, [1032].time.Hour := 11, [1032].time.Minute := 34, [1032].time.Second := 59, [1032].time.DST_ON := 1, [1033].log_data[0].min := 1.0, [1033].log_data[0].max := 1.0, [1033].log_data[0].total := 300.0, [1033].log_data[0].time := 300.0, [1033].log_data[0].minminute := 35, [1033].log_data[0].maxminute := 35, [1033].log_data[0].valid := 1, [1033].log_data[1].valid := 1, [1033].log_data[2].valid := 1, [1033].log_data[3].valid := 1, [1033].log_data[4].valid := 1, [1033].time.Year := 2022, [1033].time.Month := 4, [1033].time.Day := 27, [1033].time.Hour := 11, [1033].time.Minute := 39, [1033].time.Second := 59, [1033].time.DST_ON := 1, [1034].log_data[0].min := 1.0, [1034].log_data[0].max := 1.0, [1034].log_data[0].total := 300.0, [1034].log_data[0].time := 300.0, [1034].log_data[0].minminute := 40, [1034].log_data[0].maxminute := 40, [1034].log_data[0].valid := 1, [1034].log_data[1].valid := 1, [1034].log_data[2].valid := 1, [1034].log_data[3].valid := 1, [1034].log_data[4].valid := 1, [1034].time.Year := 2022, [1034].time.Month := 4, [1034].time.Day := 27, [1034].time.Hour := 11, [1034].time.Minute := 44, [1034].time.Second := 59, [1034].time.DST_ON := 1, [1035].log_data[0].min := 1.0, [1035].log_data[0].max := 1.0, [1035].log_data[0].total := 300.0, [1035].log_data[0].time := 300.0, [1035].log_data[0].minminute := 45,
        [1035].log_data[0].maxminute := 45, [1035].log_data[0].valid := 1, [1035].log_data[1].valid := 1, [1035].log_data[2].valid := 1, [1035].log_data[3].valid := 1, [1035].log_data[4].valid := 1, [1035].time.Year := 2022, [1035].time.Month := 4, [1035].time.Day := 27, [1035].time.Hour := 11, [1035].time.Minute := 49, [1035].time.Second := 59, [1035].time.DST_ON := 1, [1036].log_data[0].min := 1.0, [1036].log_data[0].max := 1.0, [1036].log_data[0].total := 300.0, [1036].log_data[0].time := 300.0, [1036].log_data[0].minminute := 50, [1036].log_data[0].maxminute := 50, [1036].log_data[0].valid := 1, [1036].log_data[1].valid := 1, [1036].log_data[2].valid := 1, [1036].log_data[3].valid := 1, [1036].log_data[4].valid := 1, [1036].time.Year := 2022, [1036].time.Month := 4, [1036].time.Day := 27, [1036].time.Hour := 11, [1036].time.Minute := 54, [1036].time.Second := 59, [1036].time.DST_ON := 1, [1037].log_data[0].min := 1.0, [1037].log_data[0].max := 1.0, [1037].log_data[0].total := 300.0, [1037].log_data[0].time := 300.0, [1037].log_data[0].minminute := 55, [1037].log_data[0].maxminute := 55, [1037].log_data[0].valid := 1, [1037].log_data[1].valid := 1, [1037].log_data[2].valid := 1, [1037].log_data[3].valid := 1, [1037].log_data[4].valid := 1, [1037].time.Year := 2022, [1037].time.Month := 4, [1037].time.Day := 27, [1037].time.Hour := 11, [1037].time.Minute := 59, [1037].time.Second := 59, [1037].time.DST_ON := 1, [1038].log_data[0].min := 1.0, [1038].log_data[0].max := 1.0, [1038].log_data[0].total := 300.0, [1038].log_data[0].time := 300.0, [1038].log_data[0].valid := 1, [1038].log_data[1].valid := 1, [1038].log_data[2].valid := 1, [1038].log_data[3].valid := 1, [1038].log_data[4].valid := 1, [1038].time.Year := 2022, [1038].time.Month := 4,
        [1038].time.Day := 27, [1038].time.Hour := 12, [1038].time.Minute := 4, [1038].time.Second := 59, [1038].time.DST_ON := 1, [1039].log_data[0].min := 1.0, [1039].log_data[0].max := 1.0, [1039].log_data[0].total := 300.0, [1039].log_data[0].time := 300.0, [1039].log_data[0].minminute := 5, [1039].log_data[0].maxminute := 5, [1039].log_data[0].valid := 1, [1039].log_data[1].valid := 1, [1039].log_data[2].valid := 1, [1039].log_data[3].valid := 1, [1039].log_data[4].valid := 1, [1039].time.Year := 2022, [1039].time.Month := 4, [1039].time.Day := 27, [1039].time.Hour := 12, [1039].time.Minute := 9, [1039].time.Second := 59, [1039].time.DST_ON := 1, [1040].log_data[0].min := 1.0, [1040].log_data[0].max := 1.0, [1040].log_data[0].total := 300.0, [1040].log_data[0].time := 300.0, [1040].log_data[0].minminute := 10, [1040].log_data[0].maxminute := 10, [1040].log_data[0].valid := 1, [1040].log_data[1].valid := 1, [1040].log_data[2].valid := 1, [1040].log_data[3].valid := 1, [1040].log_data[4].valid := 1, [1040].time.Year := 2022, [1040].time.Month := 4, [1040].time.Day := 27, [1040].time.Hour := 12, [1040].time.Minute := 14, [1040].time.Second := 59, [1040].time.DST_ON := 1, [1041].log_data[0].min := 1.0, [1041].log_data[0].max := 1.0, [1041].log_data[0].total := 300.0, [1041].log_data[0].time := 300.0, [1041].log_data[0].minminute := 15, [1041].log_data[0].maxminute := 15, [1041].log_data[0].valid := 1, [1041].log_data[1].valid := 1, [1041].log_data[2].valid := 1, [1041].log_data[3].valid := 1, [1041].log_data[4].valid := 1, [1041].time.Year := 2022, [1041].time.Month := 4, [1041].time.Day := 27, [1041].time.Hour := 12, [1041].time.Minute := 19, [1041].time.Second := 59, [1041].time.DST_ON := 1, [1042].log_data[0].min := 1.0,
        [1042].log_data[0].max := 1.0, [1042].log_data[0].total := 300.0, [1042].log_data[0].time := 300.0, [1042].log_data[0].minminute := 20, [1042].log_data[0].maxminute := 20, [1042].log_data[0].valid := 1, [1042].log_data[1].valid := 1, [1042].log_data[2].valid := 1, [1042].log_data[3].valid := 1, [1042].log_data[4].valid := 1, [1042].time.Year := 2022, [1042].time.Month := 4, [1042].time.Day := 27, [1042].time.Hour := 12, [1042].time.Minute := 24, [1042].time.Second := 59, [1042].time.DST_ON := 1, [1043].log_data[0].min := 1.0, [1043].log_data[0].max := 1.0, [1043].log_data[0].total := 300.0, [1043].log_data[0].time := 300.0, [1043].log_data[0].minminute := 25, [1043].log_data[0].maxminute := 25, [1043].log_data[0].valid := 1, [1043].log_data[1].valid := 1, [1043].log_data[2].valid := 1, [1043].log_data[3].valid := 1, [1043].log_data[4].valid := 1, [1043].time.Year := 2022, [1043].time.Month := 4, [1043].time.Day := 27, [1043].time.Hour := 12, [1043].time.Minute := 29, [1043].time.Second := 59, [1043].time.DST_ON := 1, [1044].log_data[0].min := 1.0, [1044].log_data[0].max := 1.0, [1044].log_data[0].total := 300.0, [1044].log_data[0].time := 300.0, [1044].log_data[0].minminute := 30, [1044].log_data[0].maxminute := 30, [1044].log_data[0].valid := 1, [1044].log_data[1].valid := 1, [1044].log_data[2].valid := 1, [1044].log_data[3].valid := 1, [1044].log_data[4].valid := 1, [1044].time.Year := 2022, [1044].time.Month := 4, [1044].time.Day := 27, [1044].time.Hour := 12, [1044].time.Minute := 34, [1044].time.Second := 59, [1044].time.DST_ON := 1, [1045].log_data[0].min := 1.0, [1045].log_data[0].max := 1.0, [1045].log_data[0].total := 300.0, [1045].log_data[0].time := 300.0, [1045].log_data[0].minminute := 35, [1045].log_data[0].maxminute := 35, [1045].log_data[0].valid := 1,
        [1045].log_data[1].valid := 1, [1045].log_data[2].valid := 1, [1045].log_data[3].valid := 1, [1045].log_data[4].valid := 1, [1045].time.Year := 2022, [1045].time.Month := 4, [1045].time.Day := 27, [1045].time.Hour := 12, [1045].time.Minute := 39, [1045].time.Second := 59, [1045].time.DST_ON := 1, [1046].log_data[0].min := 1.0, [1046].log_data[0].max := 1.0, [1046].log_data[0].total := 300.0, [1046].log_data[0].time := 300.0, [1046].log_data[0].minminute := 40, [1046].log_data[0].maxminute := 40, [1046].log_data[0].valid := 1, [1046].log_data[1].valid := 1, [1046].log_data[2].valid := 1, [1046].log_data[3].valid := 1, [1046].log_data[4].valid := 1, [1046].time.Year := 2022, [1046].time.Month := 4, [1046].time.Day := 27, [1046].time.Hour := 12, [1046].time.Minute := 44, [1046].time.Second := 59, [1046].time.DST_ON := 1, [1047].log_data[0].min := 1.0, [1047].log_data[0].max := 1.0, [1047].log_data[0].total := 300.0, [1047].log_data[0].time := 300.0, [1047].log_data[0].minminute := 45, [1047].log_data[0].maxminute := 45, [1047].log_data[0].valid := 1, [1047].log_data[1].valid := 1, [1047].log_data[2].valid := 1, [1047].log_data[3].valid := 1, [1047].log_data[4].valid := 1, [1047].time.Year := 2022, [1047].time.Month := 4, [1047].time.Day := 27, [1047].time.Hour := 12, [1047].time.Minute := 49, [1047].time.Second := 59, [1047].time.DST_ON := 1, [1048].log_data[0].min := 1.0, [1048].log_data[0].max := 1.0, [1048].log_data[0].total := 300.0, [1048].log_data[0].time := 300.0, [1048].log_data[0].minminute := 50, [1048].log_data[0].maxminute := 50, [1048].log_data[0].valid := 1, [1048].log_data[1].valid := 1, [1048].log_data[2].valid := 1, [1048].log_data[3].valid := 1, [1048].log_data[4].valid := 1, [1048].time.Year := 2022, [1048].time.Month := 4,
        [1048].time.Day := 27, [1048].time.Hour := 12, [1048].time.Minute := 54, [1048].time.Second := 59, [1048].time.DST_ON := 1, [1049].log_data[0].min := 1.0, [1049].log_data[0].max := 1.0, [1049].log_data[0].total := 300.0, [1049].log_data[0].time := 300.0, [1049].log_data[0].minminute := 55, [1049].log_data[0].maxminute := 55, [1049].log_data[0].valid := 1, [1049].log_data[1].valid := 1, [1049].log_data[2].valid := 1, [1049].log_data[3].valid := 1, [1049].log_data[4].valid := 1, [1049].time.Year := 2022, [1049].time.Month := 4, [1049].time.Day := 27, [1049].time.Hour := 12, [1049].time.Minute := 59, [1049].time.Second := 59, [1049].time.DST_ON := 1, [1050].log_data[0].min := 1.0, [1050].log_data[0].max := 1.0, [1050].log_data[0].total := 300.0, [1050].log_data[0].time := 300.0, [1050].log_data[0].valid := 1, [1050].log_data[1].valid := 1, [1050].log_data[2].valid := 1, [1050].log_data[3].valid := 1, [1050].log_data[4].valid := 1, [1050].time.Year := 2022, [1050].time.Month := 4, [1050].time.Day := 27, [1050].time.Hour := 13, [1050].time.Minute := 4, [1050].time.Second := 59, [1050].time.DST_ON := 1, [1051].log_data[0].min := 1.0, [1051].log_data[0].max := 1.0, [1051].log_data[0].total := 300.0, [1051].log_data[0].time := 300.0, [1051].log_data[0].minminute := 5, [1051].log_data[0].maxminute := 5, [1051].log_data[0].valid := 1, [1051].log_data[1].valid := 1, [1051].log_data[2].valid := 1, [1051].log_data[3].valid := 1, [1051].log_data[4].valid := 1, [1051].time.Year := 2022, [1051].time.Month := 4, [1051].time.Day := 27, [1051].time.Hour := 13, [1051].time.Minute := 9, [1051].time.Second := 59, [1051].time.DST_ON := 1, [1052].log_data[0].min := 1.0, [1052].log_data[0].max := 1.0, [1052].log_data[0].total := 300.0,
